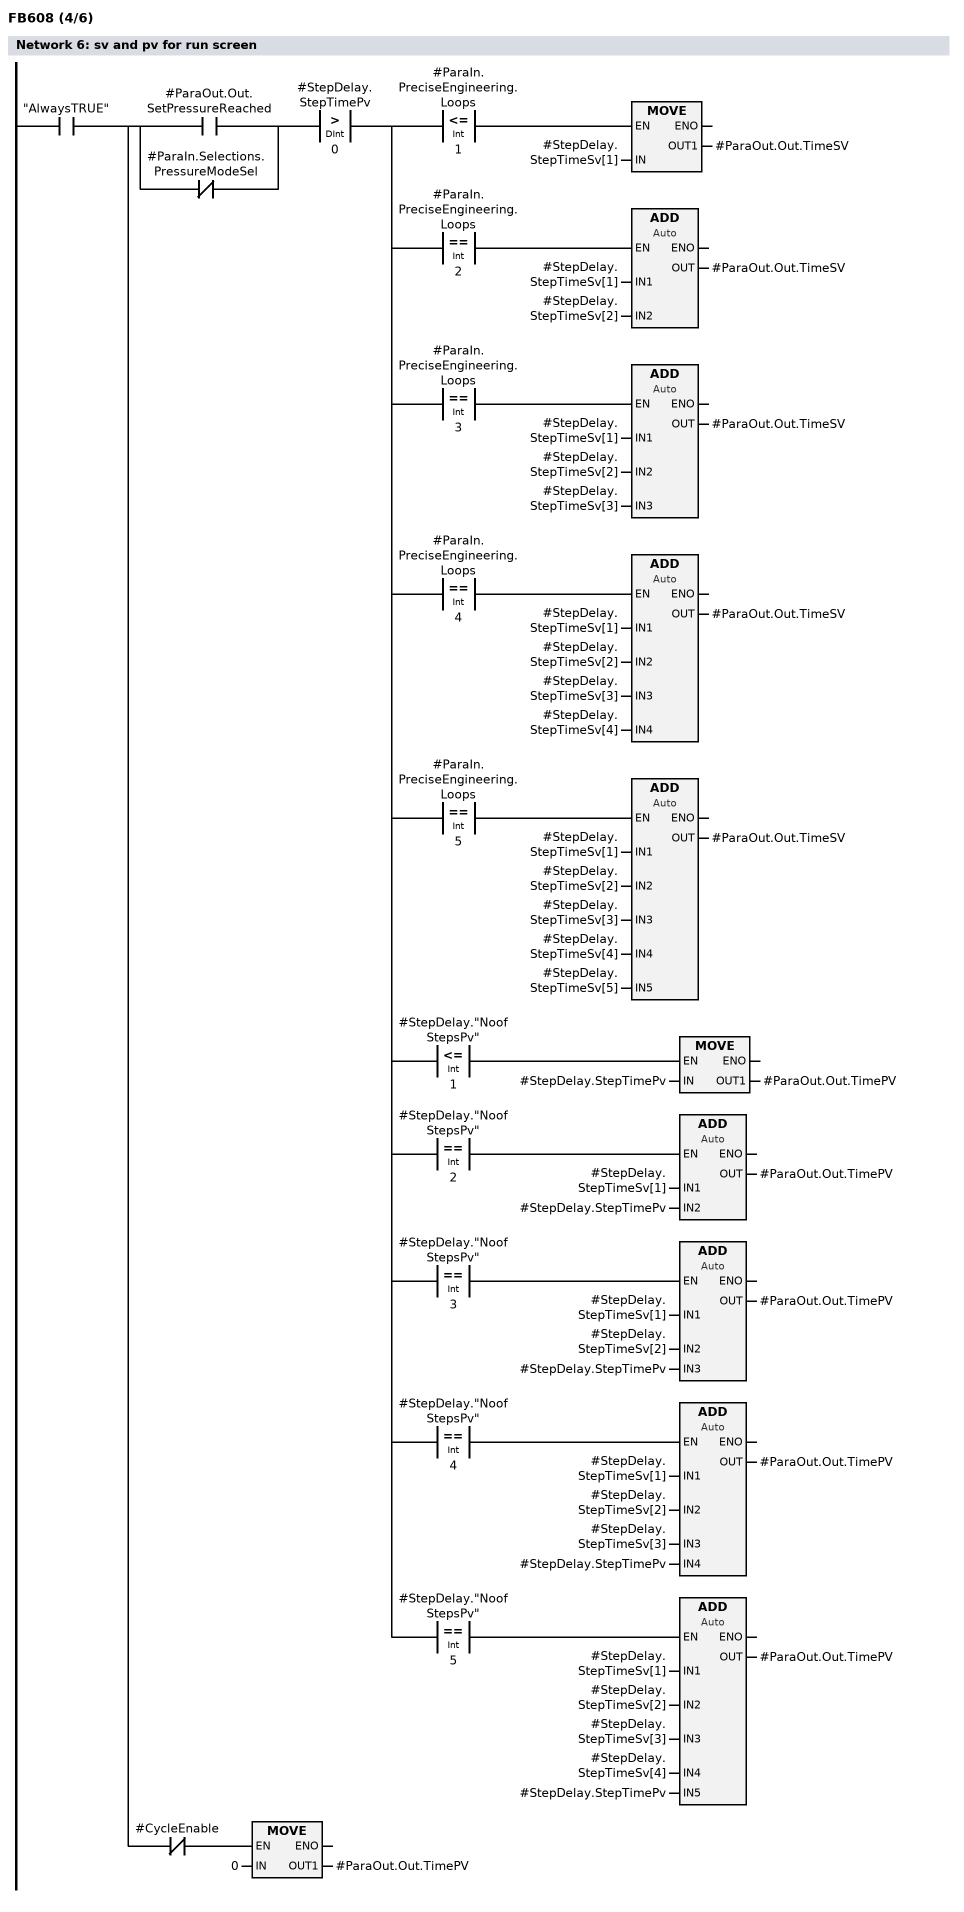
   RUNG wire#powerrail
      Contact( "AlwaysTRUE" )
      wire#w1
      Contact( #ParaOut.Out.SetPressureReached )
      wire#w2
      { S7_Templates := "SrcType := DInt" } GT_Contact(in1 := #StepDelay.StepTimePv, in2 := 0)
      wire#w3
      { S7_Templates := "SrcType := Int" } LE_Contact(in1 := #ParaIn.PreciseEngineering.Loops, in2 := 1)
      Move(in := #StepDelay.StepTimeSv[1], out1 => #ParaOut.Out.TimeSV)
   END_RUNG
   RUNG wire#w1
      I_Contact( #ParaIn.Selections.PressureModeSel )
   END_RUNG wire#w2
   RUNG wire#w3
      { S7_Templates := "SrcType := Int" } EQ_Contact(in1 := #ParaIn.PreciseEngineering.Loops, in2 := 2)
      Add(in1 := #StepDelay.StepTimeSv[1], in2 := #StepDelay.StepTimeSv[2], out => #ParaOut.Out.TimeSV)
   END_RUNG
   RUNG wire#w3
      { S7_Templates := "SrcType := Int" } EQ_Contact(in1 := #ParaIn.PreciseEngineering.Loops, in2 := 3)
      Add(in1 := #StepDelay.StepTimeSv[1], in2 := #StepDelay.StepTimeSv[2], in3 := #StepDelay.StepTimeSv[3], out => #ParaOut.Out.TimeSV)
   END_RUNG
   RUNG wire#w3
      { S7_Templates := "SrcType := Int" } EQ_Contact(in1 := #ParaIn.PreciseEngineering.Loops, in2 := 4)
      Add(in1 := #StepDelay.StepTimeSv[1], in2 := #StepDelay.StepTimeSv[2], in3 := #StepDelay.StepTimeSv[3], in4 := #StepDelay.StepTimeSv[4], out => #ParaOut.Out.TimeSV)
   END_RUNG
   RUNG wire#w3
      { S7_Templates := "SrcType := Int" } EQ_Contact(in1 := #ParaIn.PreciseEngineering.Loops, in2 := 5)
      Add(in1 := #StepDelay.StepTimeSv[1], in2 := #StepDelay.StepTimeSv[2], in3 := #StepDelay.StepTimeSv[3], in4 := #StepDelay.StepTimeSv[4], in5 := #StepDelay.StepTimeSv[5], out => #ParaOut.Out.TimeSV)
   END_RUNG
   RUNG wire#w3
      { S7_Templates := "SrcType := Int" } LE_Contact(in1 := #StepDelay."Noof StepsPv", in2 := 1)
      Move(in := #StepDelay.StepTimePv, out1 => #ParaOut.Out.TimePV)
   END_RUNG
   RUNG wire#w3
      { S7_Templates := "SrcType := Int" } EQ_Contact(in1 := #StepDelay."Noof StepsPv", in2 := 2)
      Add(in1 := #StepDelay.StepTimeSv[1], in2 := #StepDelay.StepTimePv, out => #ParaOut.Out.TimePV)
   END_RUNG
   RUNG wire#w3
      { S7_Templates := "SrcType := Int" } EQ_Contact(in1 := #StepDelay."Noof StepsPv", in2 := 3)
      Add(in1 := #StepDelay.StepTimeSv[1], in2 := #StepDelay.StepTimeSv[2], in3 := #StepDelay.StepTimePv, out => #ParaOut.Out.TimePV)
   END_RUNG
   RUNG wire#w3
      { S7_Templates := "SrcType := Int" } EQ_Contact(in1 := #StepDelay."Noof StepsPv", in2 := 4)
      Add(in1 := #StepDelay.StepTimeSv[1], in2 := #StepDelay.StepTimeSv[2], in3 := #StepDelay.StepTimeSv[3], in4 := #StepDelay.StepTimePv, out => #ParaOut.Out.TimePV)
   END_RUNG
   RUNG wire#w3
      { S7_Templates := "SrcType := Int" } EQ_Contact(in1 := #StepDelay."Noof StepsPv", in2 := 5)
      Add(in1 := #StepDelay.StepTimeSv[1], in2 := #StepDelay.StepTimeSv[2], in3 := #StepDelay.StepTimeSv[3], in4 := #StepDelay.StepTimeSv[4], in5 := #StepDelay.StepTimePv, out => #ParaOut.Out.TimePV)
   END_RUNG
   RUNG wire#w1
      I_Contact( #CycleEnable )
      Move(in := 0, out1 => #ParaOut.Out.TimePV)
   END_RUNG
   // the same network as SCL:
   #_w1 := "AlwaysTRUE" AND (#ParaOut.Out.SetPressureReached OR NOT #ParaIn.Selections.PressureModeSel) AND (#StepDelay.StepTimePv > 0);
   IF #_w1 AND (#ParaIn.PreciseEngineering.Loops <= 1) THEN
       #ParaOut.Out.TimeSV := #StepDelay.StepTimeSv[1];
   END_IF;
   IF #_w1 AND (#ParaIn.PreciseEngineering.Loops = 2) THEN
       #ParaOut.Out.TimeSV := #StepDelay.StepTimeSv[1] + #StepDelay.StepTimeSv[2];
   END_IF;
   IF #_w1 AND (#ParaIn.PreciseEngineering.Loops = 3) THEN
       #ParaOut.Out.TimeSV := #StepDelay.StepTimeSv[1] + #StepDelay.StepTimeSv[2] + #StepDelay.StepTimeSv[3];
   END_IF;
   IF #_w1 AND (#ParaIn.PreciseEngineering.Loops = 4) THEN
       #ParaOut.Out.TimeSV := #StepDelay.StepTimeSv[1] + #StepDelay.StepTimeSv[2] + #StepDelay.StepTimeSv[3] + #StepDelay.StepTimeSv[4];
   END_IF;
   IF #_w1 AND (#ParaIn.PreciseEngineering.Loops = 5) THEN
       #ParaOut.Out.TimeSV := #StepDelay.StepTimeSv[1] + #StepDelay.StepTimeSv[2] + #StepDelay.StepTimeSv[3] + #StepDelay.StepTimeSv[4] + #StepDelay.StepTimeSv[5];
   END_IF;
   IF #_w1 AND (#StepDelay."Noof StepsPv" <= 1) THEN #ParaOut.Out.TimePV := #StepDelay.StepTimePv; END_IF;
   IF #_w1 AND (#StepDelay."Noof StepsPv" = 2) THEN
       #ParaOut.Out.TimePV := #StepDelay.StepTimeSv[1] + #StepDelay.StepTimePv;
   END_IF;
   IF #_w1 AND (#StepDelay."Noof StepsPv" = 3) THEN
       #ParaOut.Out.TimePV := #StepDelay.StepTimeSv[1] + #StepDelay.StepTimeSv[2] + #StepDelay.StepTimePv;
   END_IF;
   IF #_w1 AND (#StepDelay."Noof StepsPv" = 4) THEN
       #ParaOut.Out.TimePV := #StepDelay.StepTimeSv[1] + #StepDelay.StepTimeSv[2] + #StepDelay.StepTimeSv[3] + #StepDelay.StepTimePv;
   END_IF;
   IF #_w1 AND (#StepDelay."Noof StepsPv" = 5) THEN
       #ParaOut.Out.TimePV := #StepDelay.StepTimeSv[1] + #StepDelay.StepTimeSv[2] + #StepDelay.StepTimeSv[3] + #StepDelay.StepTimeSv[4] + #StepDelay.StepTimePv;
   END_IF;
   IF "AlwaysTRUE" AND NOT #CycleEnable THEN #ParaOut.Out.TimePV := 0; END_IF;
END_REGION

REGION Network 7: #StepDelay
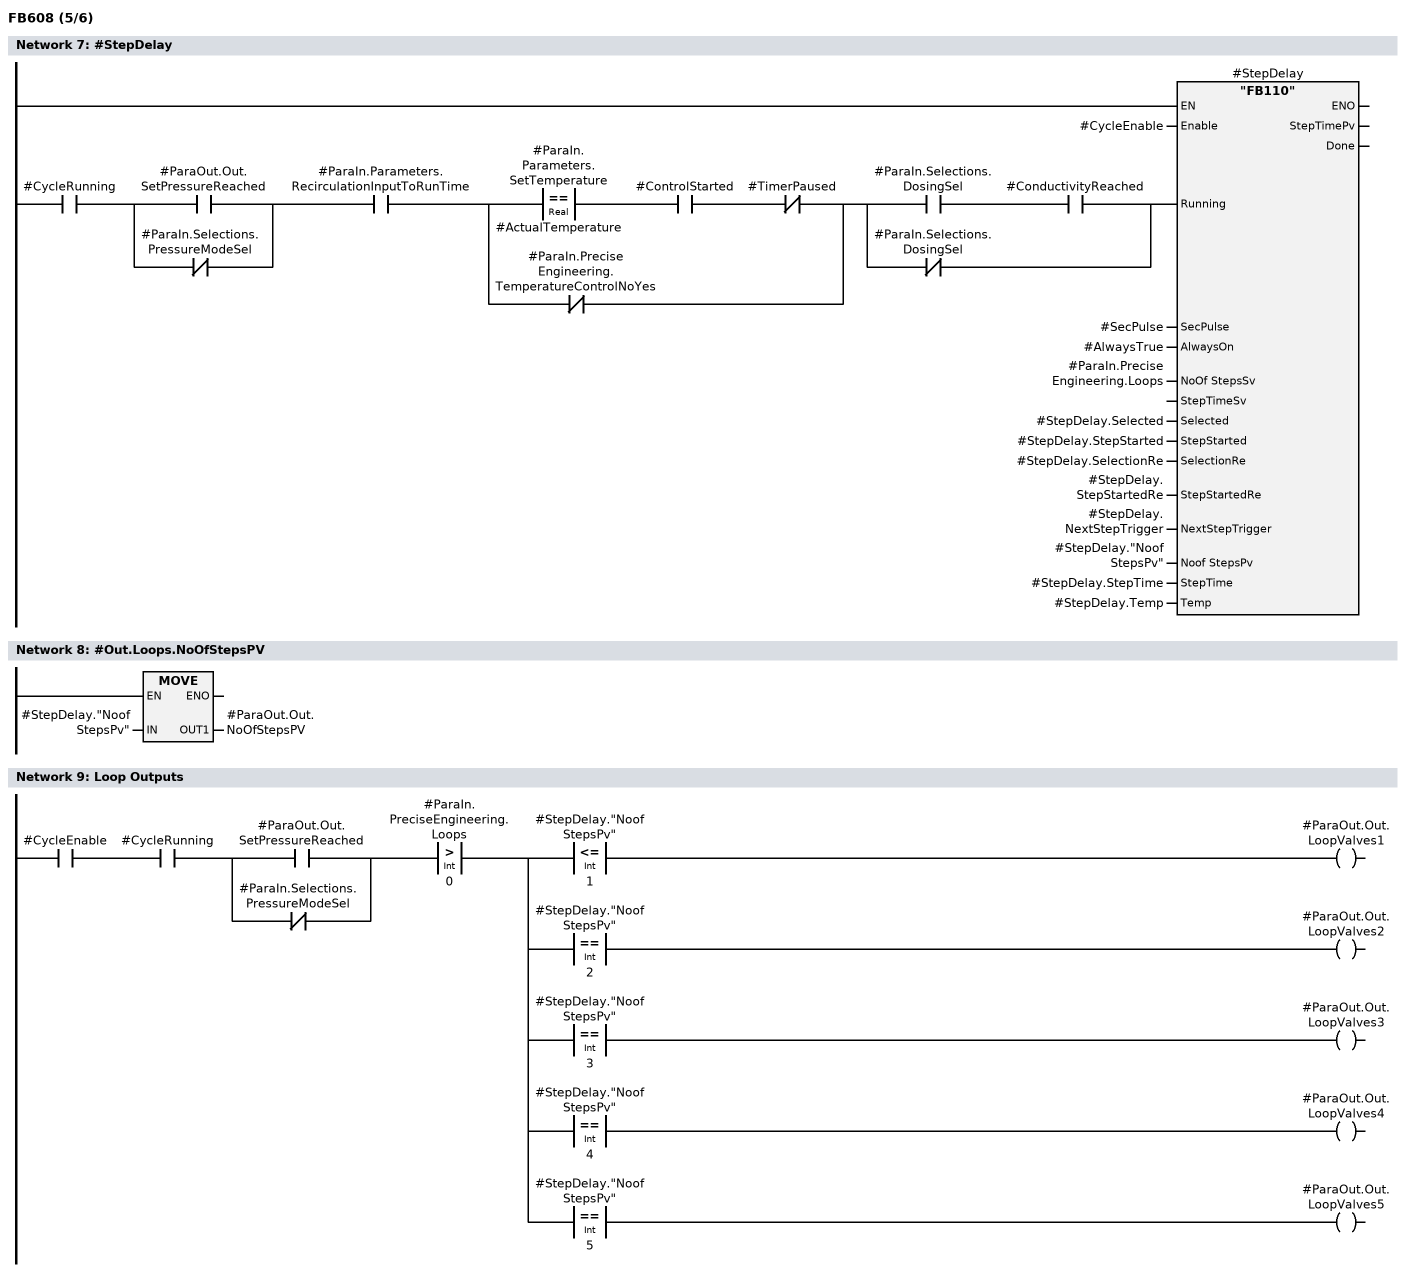
   RUNG wire#powerrail
      #StepDelay(Running := wire#w5, Enable := #CycleEnable, SecPulse := #SecPulse, AlwaysOn := #AlwaysTrue, "NoOf StepsSv" := #ParaIn.PreciseEngineering.Loops, StepTimeSv :=, Selected := #StepDelay.Selected, StepStarted := #StepDelay.StepStarted, SelectionRe := #StepDelay.SelectionRe, StepStartedRe := #StepDelay.StepStartedRe, NextStepTrigger := #StepDelay.NextStepTrigger, "Noof StepsPv" := #StepDelay."Noof StepsPv", StepTime := #StepDelay.StepTime, Temp := #StepDelay.Temp, StepTimePv =>, Done =>)
   END_RUNG
   RUNG wire#powerrail
      Contact( #CycleRunning )
      wire#w1
      Contact( #ParaOut.Out.SetPressureReached )
      wire#w2
      Contact( #ParaIn.Parameters.RecirculationInputToRunTime )
      wire#w3
      { S7_Templates := "SrcType := Real" } EQ_Contact(in1 := #ParaIn.Parameters.SetTemperature, in2 := #ActualTemperature)
      Contact( #ControlStarted )
      I_Contact( #TimerPaused )
      wire#w4
      Contact( #ParaIn.Selections.DosingSel )
      Contact( #ConductivityReached )
   END_RUNG wire#w5
   RUNG wire#w1
      I_Contact( #ParaIn.Selections.PressureModeSel )
   END_RUNG wire#w2
   RUNG wire#w3
      I_Contact( #ParaIn.PreciseEngineering.TemperatureControlNoYes )
   END_RUNG wire#w4
   RUNG wire#w4
      I_Contact( #ParaIn.Selections.DosingSel )
   END_RUNG wire#w5
   // the same network as SCL:
   #StepDelay(Enable := #CycleEnable,   // "FB110"
              Running := #CycleRunning AND (#ParaOut.Out.SetPressureReached OR NOT #ParaIn.Selections.PressureModeSel) AND #ParaIn.Parameters.RecirculationInputToRunTime AND (((#ParaIn.Parameters.SetTemperature = #ActualTemperature) AND #ControlStarted AND NOT #TimerPaused) OR NOT #ParaIn.PreciseEngineering.TemperatureControlNoYes) AND ((#ParaIn.Selections.DosingSel AND #ConductivityReached) OR NOT #ParaIn.Selections.DosingSel),
              SecPulse := #SecPulse,
              AlwaysOn := #AlwaysTrue,
              "NoOf StepsSv" := #ParaIn.PreciseEngineering.Loops,
              Selected := #StepDelay.Selected,
              StepStarted := #StepDelay.StepStarted,
              SelectionRe := #StepDelay.SelectionRe,
              StepStartedRe := #StepDelay.StepStartedRe,
              NextStepTrigger := #StepDelay.NextStepTrigger,
              "Noof StepsPv" := #StepDelay."Noof StepsPv",
              StepTime := #StepDelay.StepTime,
              Temp := #StepDelay.Temp);
END_REGION

REGION Network 8: #Out.Loops.NoOfStepsPV
   RUNG wire#powerrail
      Move(in := #StepDelay."Noof StepsPv", out1 => #ParaOut.Out.NoOfStepsPV)
   END_RUNG
   // the same network as SCL:
   #ParaOut.Out.NoOfStepsPV := #StepDelay."Noof StepsPv";
END_REGION

REGION Network 9: Loop Outputs
   RUNG wire#powerrail
      Contact( #CycleEnable )
      Contact( #CycleRunning )
      wire#w1
      Contact( #ParaOut.Out.SetPressureReached )
      wire#w2
      { S7_Templates := "SrcType := Int" } GT_Contact(in1 := #ParaIn.PreciseEngineering.Loops, in2 := 0)
      wire#w3
      { S7_Templates := "SrcType := Int" } LE_Contact(in1 := #StepDelay."Noof StepsPv", in2 := 1)
      Coil( #ParaOut.Out.LoopValves1 )
   END_RUNG
   RUNG wire#w1
      I_Contact( #ParaIn.Selections.PressureModeSel )
   END_RUNG wire#w2
   RUNG wire#w3
      { S7_Templates := "SrcType := Int" } EQ_Contact(in1 := #StepDelay."Noof StepsPv", in2 := 2)
      Coil( #ParaOut.Out.LoopValves2 )
   END_RUNG
   RUNG wire#w3
      { S7_Templates := "SrcType := Int" } EQ_Contact(in1 := #StepDelay."Noof StepsPv", in2 := 3)
      Coil( #ParaOut.Out.LoopValves3 )
   END_RUNG
   RUNG wire#w3
      { S7_Templates := "SrcType := Int" } EQ_Contact(in1 := #StepDelay."Noof StepsPv", in2 := 4)
      Coil( #ParaOut.Out.LoopValves4 )
   END_RUNG
   RUNG wire#w3
      { S7_Templates := "SrcType := Int" } EQ_Contact(in1 := #StepDelay."Noof StepsPv", in2 := 5)
      Coil( #ParaOut.Out.LoopValves5 )
   END_RUNG
   // the same network as SCL:
   #_w1 := #CycleEnable AND #CycleRunning AND (#ParaOut.Out.SetPressureReached OR NOT #ParaIn.Selections.PressureModeSel) AND (#ParaIn.PreciseEngineering.Loops > 0);
   #ParaOut.Out.LoopValves1 := #_w1 AND (#StepDelay."Noof StepsPv" <= 1);
   #ParaOut.Out.LoopValves2 := #_w1 AND (#StepDelay."Noof StepsPv" = 2);
   #ParaOut.Out.LoopValves3 := #_w1 AND (#StepDelay."Noof StepsPv" = 3);
   #ParaOut.Out.LoopValves4 := #_w1 AND (#StepDelay."Noof StepsPv" = 4);
   #ParaOut.Out.LoopValves5 := #_w1 AND (#StepDelay."Noof StepsPv" = 5);
END_REGION

REGION Network 10: Reset
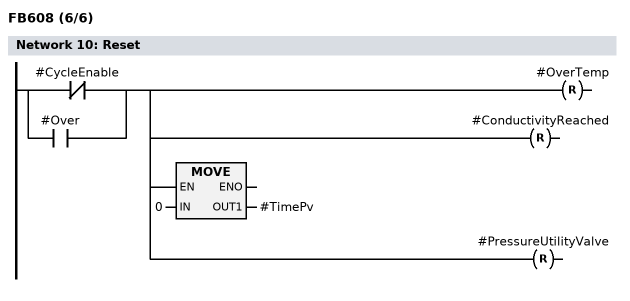
   RUNG wire#powerrail
      I_Contact( #CycleEnable )
      wire#w1
      R_Coil( #OverTemp )
   END_RUNG
   RUNG wire#powerrail
      Contact( #Over )
   END_RUNG wire#w1
   RUNG wire#w1
      R_Coil( #ConductivityReached )
   END_RUNG
   RUNG wire#w1
      { S7_GenerateENO := "TRUE" } Move(in := 0, out1 => #TimePv)
   END_RUNG
   RUNG wire#w1
      R_Coil( #PressureUtilityValve )
   END_RUNG
   // the same network as SCL:
   IF NOT #CycleEnable OR #Over THEN
       #OverTemp := FALSE;
       #ConductivityReached := FALSE;
       #TimePv := 0;
       #PressureUtilityValve := FALSE;
   END_IF;
END_REGION
END_FUNCTION_BLOCK

FUNCTION_BLOCK "FB609"   // FB609, LAD
TITLE = FB609
{ S7_Optimized_Access := 'FALSE' }
AUTHOR : PRECISE
FAMILY : PRECISE
// CIP DRAIN
// stored: AutoNumber false, SetENOAutomatically false
   VAR_INPUT
      CipSelected : Bool;
      CycleEnable : Bool;
      CycleRunning : Bool;
      SecPulse : Bool;
      AlwaysTrue : Bool;
      ParaIn : "DrainInputs";
      ActualWeight : Real;
      ActualPressure : Real;
      ActualConductivityVessel : Real;
      ActualRepetition : Int;
      ActualSkidWeight : Real;
   END_VAR
   VAR_OUTPUT
      Started : Bool;
      PressureUtilityValve : Bool;   // Air Utility
      "Line Valves" : Bool;
      ParaOut : "DrainOutputs";
      StepStatus : String[60];
      Print : "DrainPrint";
      PrintConductivityNotSampled : "ConductivityNotSampled";
   END_VAR
   VAR_IN_OUT
      Over : Bool;
      OverTemp : Bool;
      PressurePostiveTol : Real;
      PressureNegativeTol : Real;
      Temp1 : Int;
      Temp2 : Int;
      SampledConductivityVessel : Real;
      ConductivitySuccess : Bool;
      ConductivityNotSampled : Bool;
      RE1 : Bool;
      RE2 : Bool;
      RE3 : Bool;
      RE4 : Bool;
      RE5 : Bool;
      ControlStarted : Bool;
      SetPressureReached : Bool;
      DrainOverValve : Bool;
      ConductivityCheckBit : Bool;
      ActualConductivityPTL : Real;
      SampledConductivityPTL : Real;
      ConductivitySuccessVessel : Bool;
      ConductivitySuccessPtl : Bool;
      Temp3 : Int;
      Temp4 : Int;
      Temp5 : Int;
      Temp6 : Int;
      Temp7 : Int;
      Temp8 : Int;
      EndConfirmationPopupSel : Bool;
      EndConfirmationPopup : Bool;
      EndConfirmationPopupAck : Bool;
      RE_1 : Bool;
      TempBit : Bool;
      RE6 : Bool;
   END_VAR
   VAR
      ValveOnDelayPV : Int;
      ValveOffDelayPV : Int;
      StepDelay { S7_SetPoint := 'True'} : "FB110";
      ResetPrintValues { S7_SetPoint := 'True'} : TON_TIME;
   END_VAR
   // ParaIn.PreciseEngineering.Loops := 1;
   VAR_TEMP   // added for the SCL form of the ladder/FBD networks
      _w1 : Bool;
      _w2 : Bool;
      _w3 : Bool;
      _w4 : Bool;
      _w5 : Bool;
      _w6 : Bool;
      _w7 : Bool;
      _w8 : Bool;
      _w9 : Bool;
   END_VAR
BEGIN

REGION Network 1: Reset Print Status on Start
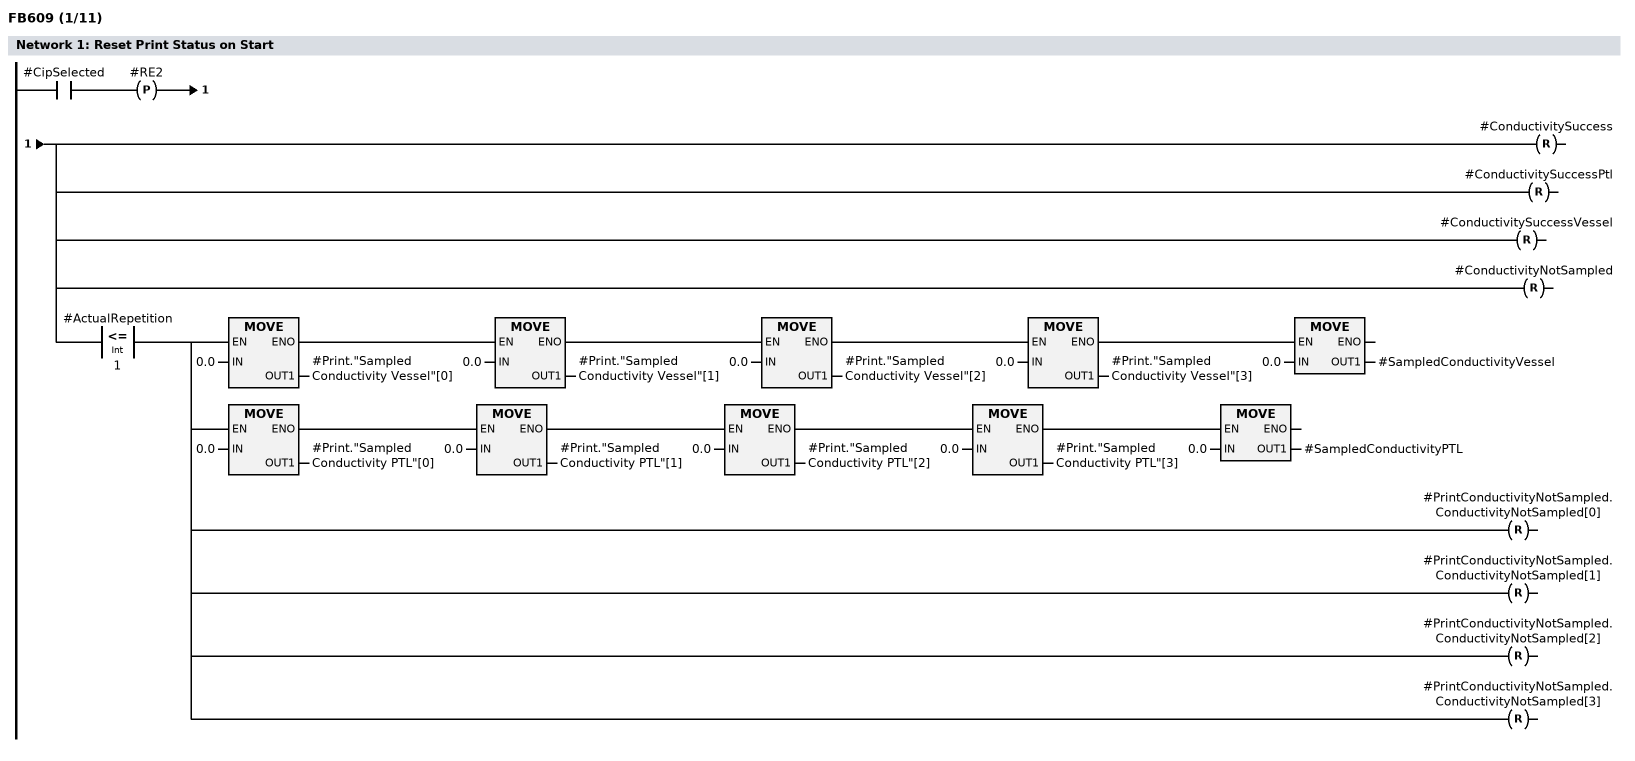
   RUNG wire#powerrail
      Contact( #CipSelected )
      P_Trig( #RE2 )
      wire#w1
      R_Coil( #ConductivitySuccess )
   END_RUNG
   RUNG wire#w1
      R_Coil( #ConductivitySuccessPtl )
   END_RUNG
   RUNG wire#w1
      R_Coil( #ConductivitySuccessVessel )
   END_RUNG
   RUNG wire#w1
      R_Coil( #ConductivityNotSampled )
   END_RUNG
   RUNG wire#w1
      { S7_Templates := "SrcType := Int" } LE_Contact(in1 := #ActualRepetition, in2 := 1)
      wire#w2
      Move(in := 0.0, out1 => #Print."SampledConductivity Vessel"[0])
      Move(in := 0.0, out1 => #Print."SampledConductivity Vessel"[1])
      Move(in := 0.0, out1 => #Print."SampledConductivity Vessel"[2])
      Move(in := 0.0, out1 => #Print."SampledConductivity Vessel"[3])
      Move(in := 0.0, out1 => #SampledConductivityVessel)
   END_RUNG
   RUNG wire#w2
      Move(in := 0.0, out1 => #Print."SampledConductivity PTL"[0])
      Move(in := 0.0, out1 => #Print."SampledConductivity PTL"[1])
      Move(in := 0.0, out1 => #Print."SampledConductivity PTL"[2])
      Move(in := 0.0, out1 => #Print."SampledConductivity PTL"[3])
      Move(in := 0.0, out1 => #SampledConductivityPTL)
   END_RUNG
   RUNG wire#w2
      R_Coil( #PrintConductivityNotSampled.ConductivityNotSampled[0] )
   END_RUNG
   RUNG wire#w2
      R_Coil( #PrintConductivityNotSampled.ConductivityNotSampled[1] )
   END_RUNG
   RUNG wire#w2
      R_Coil( #PrintConductivityNotSampled.ConductivityNotSampled[2] )
   END_RUNG
   RUNG wire#w2
      R_Coil( #PrintConductivityNotSampled.ConductivityNotSampled[3] )
   END_RUNG
   // the same network as SCL:
   #_w1 := #CipSelected AND NOT #RE2;   // rising edge
   #RE2 := #CipSelected;
   IF #_w1 THEN
       #ConductivitySuccess := FALSE;
       #ConductivitySuccessPtl := FALSE;
       #ConductivitySuccessVessel := FALSE;
       #ConductivityNotSampled := FALSE;
   END_IF;
   IF #_w1 AND (#ActualRepetition <= 1) THEN
       #Print."SampledConductivity Vessel"[0] := 0.0;
       #Print."SampledConductivity Vessel"[1] := 0.0;
       #Print."SampledConductivity Vessel"[2] := 0.0;
       #Print."SampledConductivity Vessel"[3] := 0.0;
       #SampledConductivityVessel := 0.0;
       #Print."SampledConductivity PTL"[0] := 0.0;
       #Print."SampledConductivity PTL"[1] := 0.0;
       #Print."SampledConductivity PTL"[2] := 0.0;
       #Print."SampledConductivity PTL"[3] := 0.0;
       #SampledConductivityPTL := 0.0;
       #PrintConductivityNotSampled.ConductivityNotSampled[0] := FALSE;
       #PrintConductivityNotSampled.ConductivityNotSampled[1] := FALSE;
       #PrintConductivityNotSampled.ConductivityNotSampled[2] := FALSE;
       #PrintConductivityNotSampled.ConductivityNotSampled[3] := FALSE;
   END_IF;
END_REGION

REGION Network 2: Drain Started
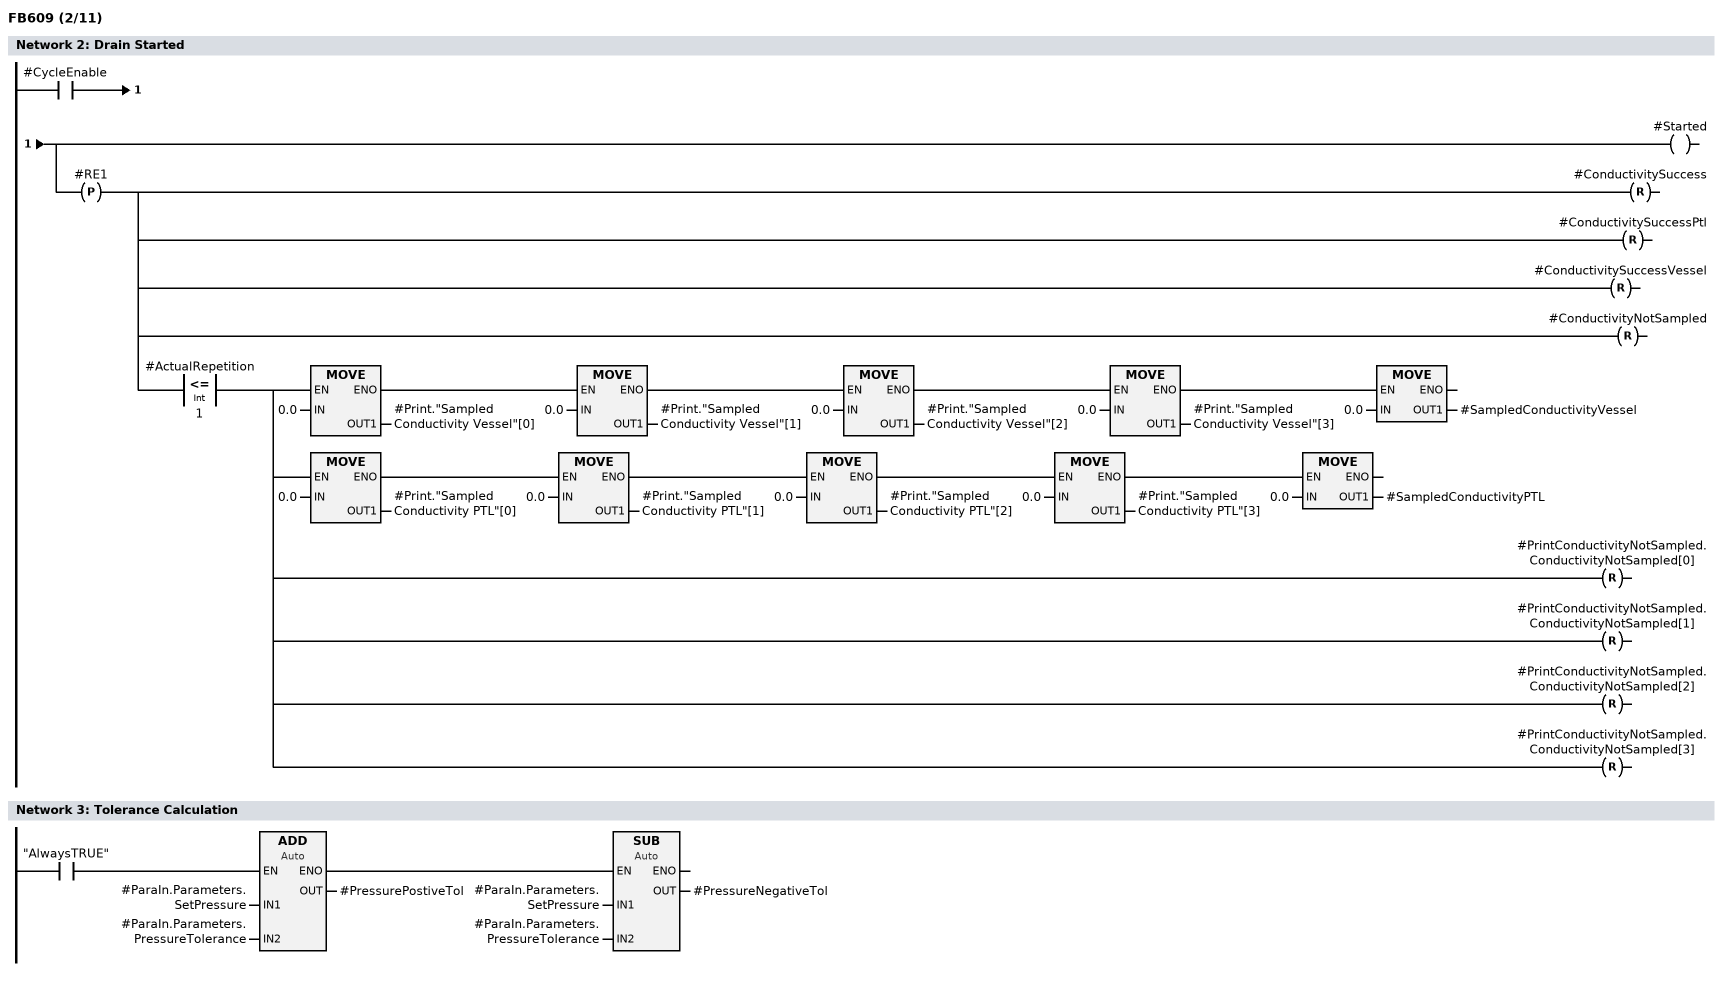
   RUNG wire#powerrail
      Contact( #CycleEnable )
      wire#w1
      Coil( #Started )
   END_RUNG
   RUNG wire#w1
      P_Trig( #RE1 )
      wire#w2
      R_Coil( #ConductivitySuccess )
   END_RUNG
   RUNG wire#w2
      R_Coil( #ConductivitySuccessPtl )
   END_RUNG
   RUNG wire#w2
      R_Coil( #ConductivitySuccessVessel )
   END_RUNG
   RUNG wire#w2
      R_Coil( #ConductivityNotSampled )
   END_RUNG
   RUNG wire#w2
      { S7_Templates := "SrcType := Int" } LE_Contact(in1 := #ActualRepetition, in2 := 1)
      wire#w3
      Move(in := 0.0, out1 => #Print."SampledConductivity Vessel"[0])
      Move(in := 0.0, out1 => #Print."SampledConductivity Vessel"[1])
      Move(in := 0.0, out1 => #Print."SampledConductivity Vessel"[2])
      Move(in := 0.0, out1 => #Print."SampledConductivity Vessel"[3])
      Move(in := 0.0, out1 => #SampledConductivityVessel)
   END_RUNG
   RUNG wire#w3
      Move(in := 0.0, out1 => #Print."SampledConductivity PTL"[0])
      Move(in := 0.0, out1 => #Print."SampledConductivity PTL"[1])
      Move(in := 0.0, out1 => #Print."SampledConductivity PTL"[2])
      Move(in := 0.0, out1 => #Print."SampledConductivity PTL"[3])
      Move(in := 0.0, out1 => #SampledConductivityPTL)
   END_RUNG
   RUNG wire#w3
      R_Coil( #PrintConductivityNotSampled.ConductivityNotSampled[0] )
   END_RUNG
   RUNG wire#w3
      R_Coil( #PrintConductivityNotSampled.ConductivityNotSampled[1] )
   END_RUNG
   RUNG wire#w3
      R_Coil( #PrintConductivityNotSampled.ConductivityNotSampled[2] )
   END_RUNG
   RUNG wire#w3
      R_Coil( #PrintConductivityNotSampled.ConductivityNotSampled[3] )
   END_RUNG
   // the same network as SCL:
   #Started := #CycleEnable;
   #_w1 := #CycleEnable AND NOT #RE1;   // rising edge
   #RE1 := #CycleEnable;
   IF #_w1 THEN
       #ConductivitySuccess := FALSE;
       #ConductivitySuccessPtl := FALSE;
       #ConductivitySuccessVessel := FALSE;
       #ConductivityNotSampled := FALSE;
   END_IF;
   IF #_w1 AND (#ActualRepetition <= 1) THEN
       #Print."SampledConductivity Vessel"[0] := 0.0;
       #Print."SampledConductivity Vessel"[1] := 0.0;
       #Print."SampledConductivity Vessel"[2] := 0.0;
       #Print."SampledConductivity Vessel"[3] := 0.0;
       #SampledConductivityVessel := 0.0;
       #Print."SampledConductivity PTL"[0] := 0.0;
       #Print."SampledConductivity PTL"[1] := 0.0;
       #Print."SampledConductivity PTL"[2] := 0.0;
       #Print."SampledConductivity PTL"[3] := 0.0;
       #SampledConductivityPTL := 0.0;
       #PrintConductivityNotSampled.ConductivityNotSampled[0] := FALSE;
       #PrintConductivityNotSampled.ConductivityNotSampled[1] := FALSE;
       #PrintConductivityNotSampled.ConductivityNotSampled[2] := FALSE;
       #PrintConductivityNotSampled.ConductivityNotSampled[3] := FALSE;
   END_IF;
END_REGION

REGION Network 3: Tolerance Calculation
   RUNG wire#powerrail
      Contact( "AlwaysTRUE" )
      Add(in1 := #ParaIn.Parameters.SetPressure, in2 := #ParaIn.Parameters.PressureTolerance, out => #PressurePostiveTol)
      Sub(in1 := #ParaIn.Parameters.SetPressure, in2 := #ParaIn.Parameters.PressureTolerance, out => #PressureNegativeTol)
   END_RUNG
   // the same network as SCL:
   IF "AlwaysTRUE" THEN
       #PressurePostiveTol := #ParaIn.Parameters.SetPressure + #ParaIn.Parameters.PressureTolerance;
       #PressureNegativeTol := #ParaIn.Parameters.SetPressure - #ParaIn.Parameters.PressureTolerance;
   END_IF;
END_REGION

REGION Network 4: Logic for Output
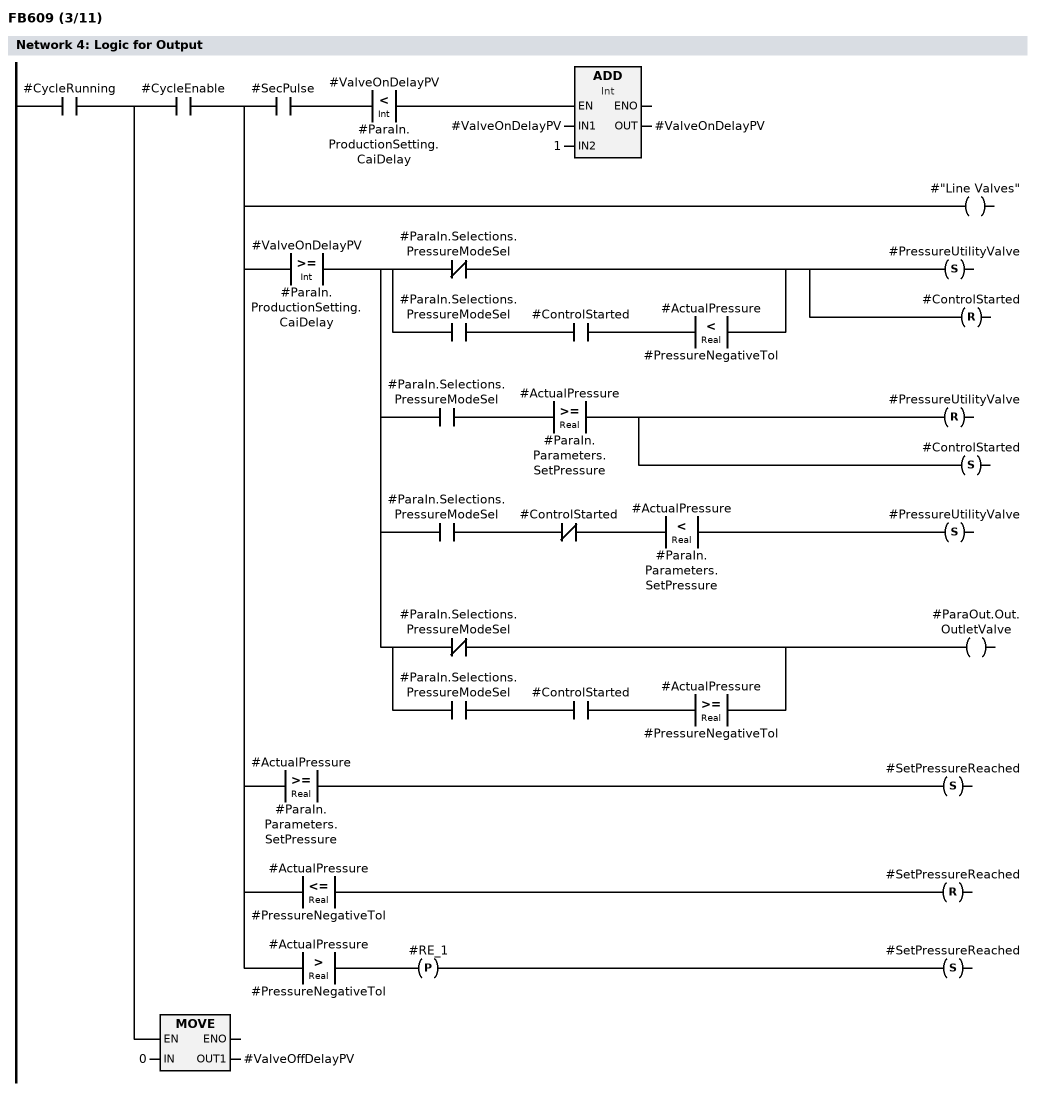
   RUNG wire#powerrail
      Contact( #CycleRunning )
      wire#w1
      Contact( #CycleEnable )
      wire#w2
      Contact( #SecPulse )
      { S7_Templates := "SrcType := Int" } LT_Contact(in1 := #ValveOnDelayPV, in2 := #ParaIn.ProductionSetting.CaiDelay)
      { S7_Templates := "SrcType := Int"; S7_GenerateENO := "TRUE" } Add(in1 := #ValveOnDelayPV, in2 := 1, out => #ValveOnDelayPV)
   END_RUNG
   RUNG wire#w2
      Coil( #"Line Valves" )
   END_RUNG
   RUNG wire#w2
      { S7_Templates := "SrcType := Int" } GE_Contact(in1 := #ValveOnDelayPV, in2 := #ParaIn.ProductionSetting.CaiDelay)
      wire#w3
      I_Contact( #ParaIn.Selections.PressureModeSel )
      wire#w4
      S_Coil( #PressureUtilityValve )
   END_RUNG
   RUNG wire#w3
      Contact( #ParaIn.Selections.PressureModeSel )
      Contact( #ControlStarted )
      { S7_Templates := "SrcType := Real" } LT_Contact(in1 := #ActualPressure, in2 := #PressureNegativeTol)
   END_RUNG wire#w4
   RUNG wire#w4
      R_Coil( #ControlStarted )
   END_RUNG
   RUNG wire#w3
      Contact( #ParaIn.Selections.PressureModeSel )
      { S7_Templates := "SrcType := Real" } GE_Contact(in1 := #ActualPressure, in2 := #ParaIn.Parameters.SetPressure)
      wire#w5
      R_Coil( #PressureUtilityValve )
   END_RUNG
   RUNG wire#w5
      S_Coil( #ControlStarted )
   END_RUNG
   RUNG wire#w3
      Contact( #ParaIn.Selections.PressureModeSel )
      I_Contact( #ControlStarted )
      { S7_Templates := "SrcType := Real" } LT_Contact(in1 := #ActualPressure, in2 := #ParaIn.Parameters.SetPressure)
      S_Coil( #PressureUtilityValve )
   END_RUNG
   RUNG wire#w3
      I_Contact( #ParaIn.Selections.PressureModeSel )
      wire#w6
      Coil( #ParaOut.Out.OutletValve )
   END_RUNG
   RUNG wire#w3
      Contact( #ParaIn.Selections.PressureModeSel )
      Contact( #ControlStarted )
      { S7_Templates := "SrcType := Real" } GE_Contact(in1 := #ActualPressure, in2 := #PressureNegativeTol)
   END_RUNG wire#w6
   RUNG wire#w2
      { S7_Templates := "SrcType := Real" } GE_Contact(in1 := #ActualPressure, in2 := #ParaIn.Parameters.SetPressure)
      S_Coil( #SetPressureReached )
   END_RUNG
   RUNG wire#w2
      { S7_Templates := "SrcType := Real" } LE_Contact(in1 := #ActualPressure, in2 := #PressureNegativeTol)
      R_Coil( #SetPressureReached )
   END_RUNG
   RUNG wire#w2
      { S7_Templates := "SrcType := Real" } GT_Contact(in1 := #ActualPressure, in2 := #PressureNegativeTol)
      P_Trig( #RE_1 )
      S_Coil( #SetPressureReached )
   END_RUNG
   RUNG wire#w1
      { S7_GenerateENO := "TRUE" } Move(in := 0, out1 => #ValveOffDelayPV)
   END_RUNG
   // the same network as SCL:
   #_w1 := #CycleRunning AND #CycleEnable;
   IF #_w1 AND #SecPulse AND (#ValveOnDelayPV < #ParaIn.ProductionSetting.CaiDelay) THEN
       #ValveOnDelayPV := #ValveOnDelayPV + 1;
   END_IF;
   #"Line Valves" := #_w1;
   #_w2 := #_w1 AND (#ValveOnDelayPV >= #ParaIn.ProductionSetting.CaiDelay);
   IF #_w2 AND (NOT #ParaIn.Selections.PressureModeSel OR (#ParaIn.Selections.PressureModeSel AND #ControlStarted AND (#ActualPressure < #PressureNegativeTol))) THEN
       #PressureUtilityValve := TRUE;
       #ControlStarted := FALSE;
   END_IF;
   IF #_w2 AND #ParaIn.Selections.PressureModeSel AND (#ActualPressure >= #ParaIn.Parameters.SetPressure) THEN
       #PressureUtilityValve := FALSE;
       #ControlStarted := TRUE;
   END_IF;
   IF #_w2 AND #ParaIn.Selections.PressureModeSel AND NOT #ControlStarted AND (#ActualPressure < #ParaIn.Parameters.SetPressure) THEN
       #PressureUtilityValve := TRUE;
   END_IF;
   #ParaOut.Out.OutletValve := #_w2 AND (NOT #ParaIn.Selections.PressureModeSel OR (#ParaIn.Selections.PressureModeSel AND #ControlStarted AND (#ActualPressure >= #PressureNegativeTol)));
   IF #_w1 AND (#ActualPressure >= #ParaIn.Parameters.SetPressure) THEN #SetPressureReached := TRUE; END_IF;
   IF #_w1 AND (#ActualPressure <= #PressureNegativeTol) THEN #SetPressureReached := FALSE; END_IF;
   #_w3 := #_w1 AND (#ActualPressure > #PressureNegativeTol);
   #_w4 := #_w3 AND NOT #RE_1;   // rising edge
   #RE_1 := #_w3;
   IF #_w4 THEN #SetPressureReached := TRUE; END_IF;
   IF #CycleRunning THEN #ValveOffDelayPV := 0; END_IF;
END_REGION

REGION Network 5: Drain Over Condition
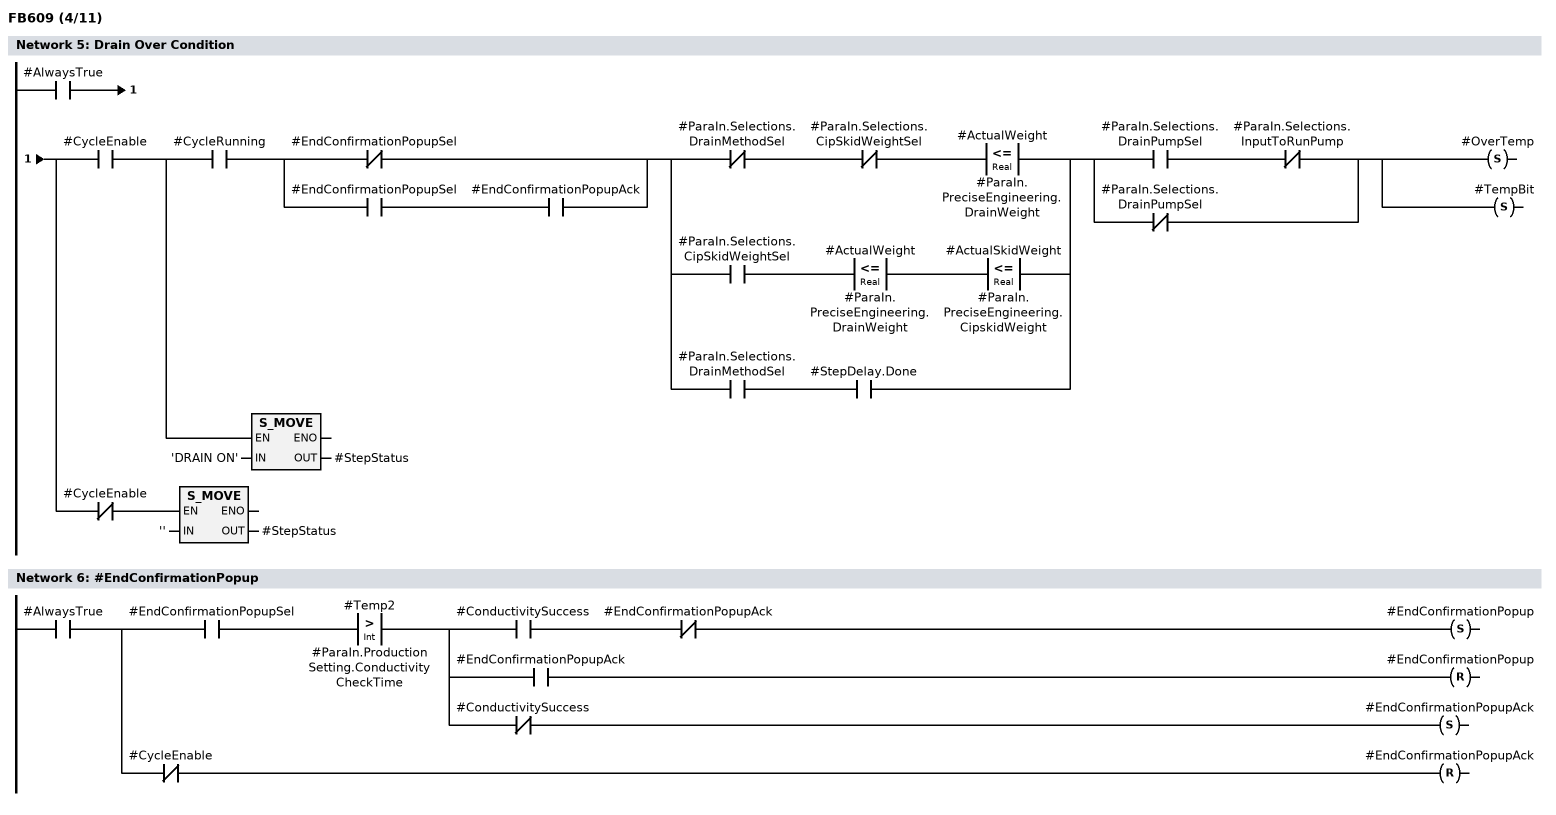
   RUNG wire#powerrail
      Contact( #AlwaysTrue )
      wire#w1
      Contact( #CycleEnable )
      wire#w2
      Contact( #CycleRunning )
      wire#w3
      I_Contact( #EndConfirmationPopupSel )
      wire#w4
      I_Contact( #ParaIn.Selections.DrainMethodSel )
      I_Contact( #ParaIn.Selections.CipSkidWeightSel )
      { S7_Templates := "SrcType := Real" } LE_Contact(in1 := #ActualWeight, in2 := #ParaIn.PreciseEngineering.DrainWeight)
      wire#w5
      Contact( #ParaIn.Selections.DrainPumpSel )
      I_Contact( #ParaIn.Selections.InputToRunPump )
      wire#w6
      S_Coil( #OverTemp )
   END_RUNG
   RUNG wire#w3
      Contact( #EndConfirmationPopupSel )
      Contact( #EndConfirmationPopupAck )
   END_RUNG wire#w4
   RUNG wire#w4
      Contact( #ParaIn.Selections.CipSkidWeightSel )
      { S7_Templates := "SrcType := Real" } LE_Contact(in1 := #ActualWeight, in2 := #ParaIn.PreciseEngineering.DrainWeight)
      { S7_Templates := "SrcType := Real" } LE_Contact(in1 := #ActualSkidWeight, in2 := #ParaIn.PreciseEngineering.CipskidWeight)
   END_RUNG wire#w5
   RUNG wire#w4
      Contact( #ParaIn.Selections.DrainMethodSel )
      Contact( #StepDelay.Done )
   END_RUNG wire#w5
   RUNG wire#w5
      I_Contact( #ParaIn.Selections.DrainPumpSel )
   END_RUNG wire#w6
   RUNG wire#w6
      S_Coil( #TempBit )
   END_RUNG
   RUNG wire#w2
      S_Move(in := 'DRAIN ON', out => #StepStatus)
   END_RUNG
   RUNG wire#w1
      I_Contact( #CycleEnable )
      S_Move(in := '', out => #StepStatus)
   END_RUNG
   // the same network as SCL:
   #_w1 := #AlwaysTrue AND #CycleEnable;
   IF #_w1 AND #CycleRunning AND (NOT #EndConfirmationPopupSel OR (#EndConfirmationPopupSel AND #EndConfirmationPopupAck)) AND ((NOT #ParaIn.Selections.DrainMethodSel AND NOT #ParaIn.Selections.CipSkidWeightSel AND (#ActualWeight <= #ParaIn.PreciseEngineering.DrainWeight)) OR (#ParaIn.Selections.CipSkidWeightSel AND (#ActualWeight <= #ParaIn.PreciseEngineering.DrainWeight) AND (#ActualSkidWeight <= #ParaIn.PreciseEngineering.CipskidWeight)) OR (#ParaIn.Selections.DrainMethodSel AND #StepDelay.Done)) AND ((#ParaIn.Selections.DrainPumpSel AND NOT #ParaIn.Selections.InputToRunPump) OR NOT #ParaIn.Selections.DrainPumpSel) THEN
       #OverTemp := TRUE;
       #TempBit := TRUE;
   END_IF;
   IF #_w1 THEN #StepStatus := 'DRAIN ON'; END_IF;
   IF #AlwaysTrue AND NOT #CycleEnable THEN #StepStatus := ''; END_IF;
END_REGION

REGION Network 6: #EndConfirmationPopup
   RUNG wire#powerrail
      Contact( #AlwaysTrue )
      wire#w1
      Contact( #EndConfirmationPopupSel )
      { S7_Templates := "SrcType := Int" } GT_Contact(in1 := #Temp2, in2 := #ParaIn.ProductionSetting.ConductivityCheckTime)
      wire#w2
      Contact( #ConductivitySuccess )
      I_Contact( #EndConfirmationPopupAck )
      S_Coil( #EndConfirmationPopup )
   END_RUNG
   RUNG wire#w2
      Contact( #EndConfirmationPopupAck )
      R_Coil( #EndConfirmationPopup )
   END_RUNG
   RUNG wire#w2
      I_Contact( #ConductivitySuccess )
      S_Coil( #EndConfirmationPopupAck )
   END_RUNG
   RUNG wire#w1
      I_Contact( #CycleEnable )
      R_Coil( #EndConfirmationPopupAck )
   END_RUNG
   // the same network as SCL:
   #_w1 := #AlwaysTrue AND #EndConfirmationPopupSel AND (#Temp2 > #ParaIn.ProductionSetting.ConductivityCheckTime);
   IF #_w1 AND #ConductivitySuccess AND NOT #EndConfirmationPopupAck THEN
       #EndConfirmationPopup := TRUE;
   END_IF;
   IF #_w1 AND #EndConfirmationPopupAck THEN #EndConfirmationPopup := FALSE; END_IF;
   IF #_w1 AND NOT #ConductivitySuccess THEN #EndConfirmationPopupAck := TRUE; END_IF;
   IF #AlwaysTrue AND NOT #CycleEnable THEN #EndConfirmationPopupAck := FALSE; END_IF;
END_REGION

REGION Network 7: Air Purge Over
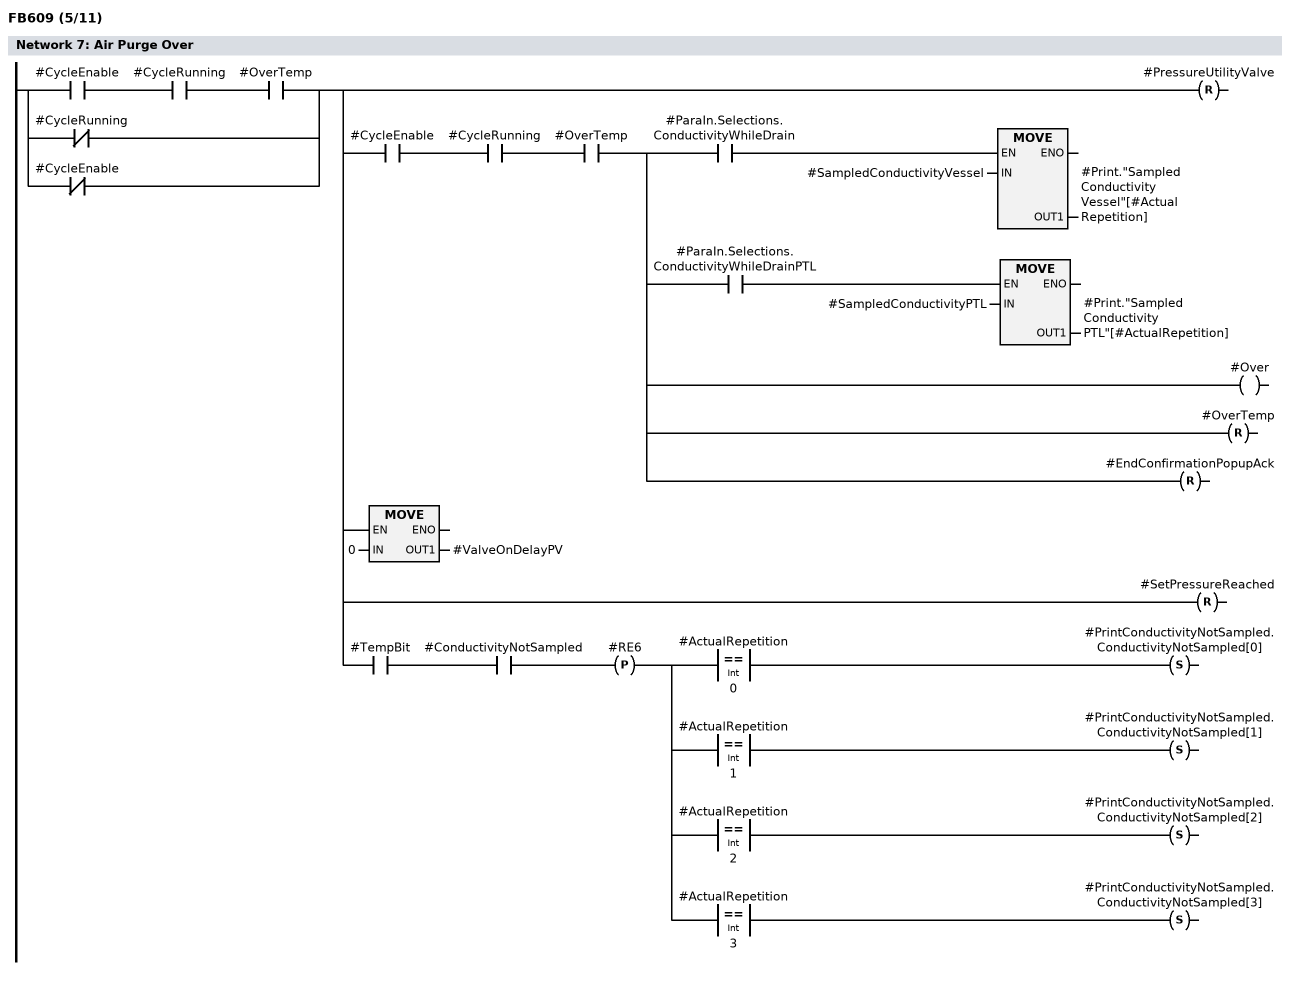
   RUNG wire#powerrail
      Contact( #CycleEnable )
      Contact( #CycleRunning )
      Contact( #OverTemp )
      wire#w1
      R_Coil( #PressureUtilityValve )
   END_RUNG
   RUNG wire#powerrail
      I_Contact( #CycleRunning )
   END_RUNG wire#w1
   RUNG wire#powerrail
      I_Contact( #CycleEnable )
   END_RUNG wire#w1
   RUNG wire#w1
      Contact( #CycleEnable )
      Contact( #CycleRunning )
      Contact( #OverTemp )
      wire#w2
      Contact( #ParaIn.Selections.ConductivityWhileDrain )
      Move(in := #SampledConductivityVessel, out1 => #Print."SampledConductivity Vessel"[#ActualRepetition])
   END_RUNG
   RUNG wire#w2
      Contact( #ParaIn.Selections.ConductivityWhileDrainPTL )
      Move(in := #SampledConductivityPTL, out1 => #Print."SampledConductivity PTL"[#ActualRepetition])
   END_RUNG
   RUNG wire#w2
      Coil( #Over )
   END_RUNG
   RUNG wire#w2
      R_Coil( #OverTemp )
   END_RUNG
   RUNG wire#w2
      R_Coil( #EndConfirmationPopupAck )
   END_RUNG
   RUNG wire#w1
      Move(in := 0, out1 => #ValveOnDelayPV)
   END_RUNG
   RUNG wire#w1
      R_Coil( #SetPressureReached )
   END_RUNG
   RUNG wire#w1
      Contact( #TempBit )
      Contact( #ConductivityNotSampled )
      P_Trig( #RE6 )
      wire#w3
      { S7_Templates := "SrcType := Int" } EQ_Contact(in1 := #ActualRepetition, in2 := 0)
      S_Coil( #PrintConductivityNotSampled.ConductivityNotSampled[0] )
   END_RUNG
   RUNG wire#w3
      { S7_Templates := "SrcType := Int" } EQ_Contact(in1 := #ActualRepetition, in2 := 1)
      S_Coil( #PrintConductivityNotSampled.ConductivityNotSampled[1] )
   END_RUNG
   RUNG wire#w3
      { S7_Templates := "SrcType := Int" } EQ_Contact(in1 := #ActualRepetition, in2 := 2)
      S_Coil( #PrintConductivityNotSampled.ConductivityNotSampled[2] )
   END_RUNG
   RUNG wire#w3
      { S7_Templates := "SrcType := Int" } EQ_Contact(in1 := #ActualRepetition, in2 := 3)
      S_Coil( #PrintConductivityNotSampled.ConductivityNotSampled[3] )
   END_RUNG
   // the same network as SCL:
   #_w1 := (#CycleEnable AND #CycleRunning AND #OverTemp) OR NOT #CycleRunning OR NOT #CycleEnable;
   IF #_w1 THEN #PressureUtilityValve := FALSE; END_IF;
   #_w2 := #_w1 AND #CycleEnable AND #CycleRunning AND #OverTemp;
   IF #_w2 AND #ParaIn.Selections.ConductivityWhileDrain THEN
       #Print."SampledConductivity Vessel"[#ActualRepetition] := #SampledConductivityVessel;
   END_IF;
   IF #_w2 AND #ParaIn.Selections.ConductivityWhileDrainPTL THEN
       #Print."SampledConductivity PTL"[#ActualRepetition] := #SampledConductivityPTL;
   END_IF;
   #Over := #_w2;
   IF #_w2 THEN
       #OverTemp := FALSE;
       #EndConfirmationPopupAck := FALSE;
   END_IF;
   IF #_w1 THEN
       #ValveOnDelayPV := 0;
       #SetPressureReached := FALSE;
   END_IF;
   #_w3 := #_w1 AND #TempBit AND #ConductivityNotSampled;
   #_w4 := #_w3 AND NOT #RE6;   // rising edge
   #RE6 := #_w3;
   IF #_w4 AND (#ActualRepetition = 0) THEN
       #PrintConductivityNotSampled.ConductivityNotSampled[0] := TRUE;
   END_IF;
   IF #_w4 AND (#ActualRepetition = 1) THEN
       #PrintConductivityNotSampled.ConductivityNotSampled[1] := TRUE;
   END_IF;
   IF #_w4 AND (#ActualRepetition = 2) THEN
       #PrintConductivityNotSampled.ConductivityNotSampled[2] := TRUE;
   END_IF;
   IF #_w4 AND (#ActualRepetition = 3) THEN
       #PrintConductivityNotSampled.ConductivityNotSampled[3] := TRUE;
   END_IF;
END_REGION

REGION Network 8: StepDelay.StepTimeSV
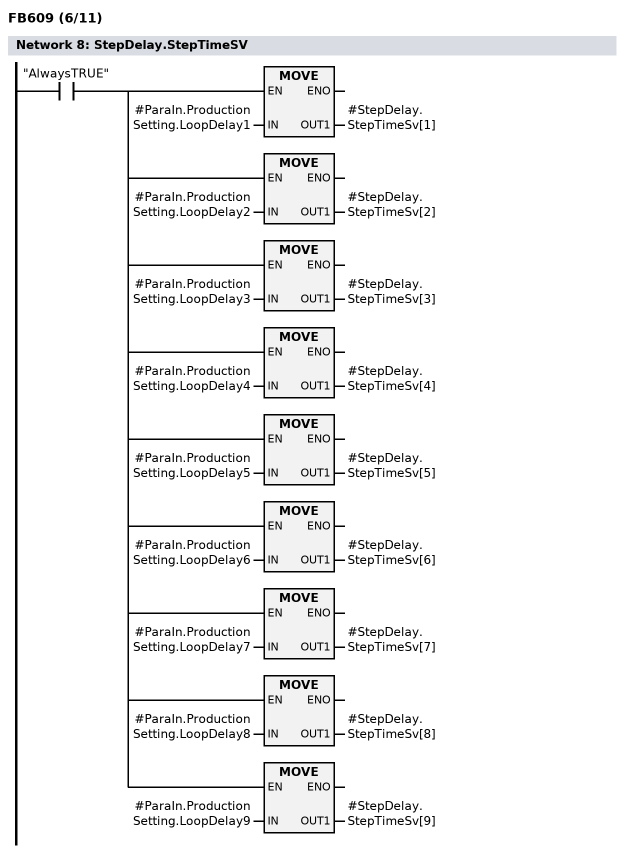
   RUNG wire#powerrail
      Contact( "AlwaysTRUE" )
      wire#w1
      Move(in := #ParaIn.ProductionSetting.LoopDelay1, out1 => #StepDelay.StepTimeSv[1])
   END_RUNG
   RUNG wire#w1
      Move(in := #ParaIn.ProductionSetting.LoopDelay2, out1 => #StepDelay.StepTimeSv[2])
   END_RUNG
   RUNG wire#w1
      Move(in := #ParaIn.ProductionSetting.LoopDelay3, out1 => #StepDelay.StepTimeSv[3])
   END_RUNG
   RUNG wire#w1
      Move(in := #ParaIn.ProductionSetting.LoopDelay4, out1 => #StepDelay.StepTimeSv[4])
   END_RUNG
   RUNG wire#w1
      Move(in := #ParaIn.ProductionSetting.LoopDelay5, out1 => #StepDelay.StepTimeSv[5])
   END_RUNG
   RUNG wire#w1
      Move(in := #ParaIn.ProductionSetting.LoopDelay6, out1 => #StepDelay.StepTimeSv[6])
   END_RUNG
   RUNG wire#w1
      Move(in := #ParaIn.ProductionSetting.LoopDelay7, out1 => #StepDelay.StepTimeSv[7])
   END_RUNG
   RUNG wire#w1
      Move(in := #ParaIn.ProductionSetting.LoopDelay8, out1 => #StepDelay.StepTimeSv[8])
   END_RUNG
   RUNG wire#w1
      Move(in := #ParaIn.ProductionSetting.LoopDelay9, out1 => #StepDelay.StepTimeSv[9])
   END_RUNG
   // the same network as SCL:
   IF "AlwaysTRUE" THEN
       #StepDelay.StepTimeSv[1] := #ParaIn.ProductionSetting.LoopDelay1;
       #StepDelay.StepTimeSv[2] := #ParaIn.ProductionSetting.LoopDelay2;
       #StepDelay.StepTimeSv[3] := #ParaIn.ProductionSetting.LoopDelay3;
       #StepDelay.StepTimeSv[4] := #ParaIn.ProductionSetting.LoopDelay4;
       #StepDelay.StepTimeSv[5] := #ParaIn.ProductionSetting.LoopDelay5;
       #StepDelay.StepTimeSv[6] := #ParaIn.ProductionSetting.LoopDelay6;
       #StepDelay.StepTimeSv[7] := #ParaIn.ProductionSetting.LoopDelay7;
       #StepDelay.StepTimeSv[8] := #ParaIn.ProductionSetting.LoopDelay8;
       #StepDelay.StepTimeSv[9] := #ParaIn.ProductionSetting.LoopDelay9;
   END_IF;
END_REGION

REGION Network 9: #StepDelay
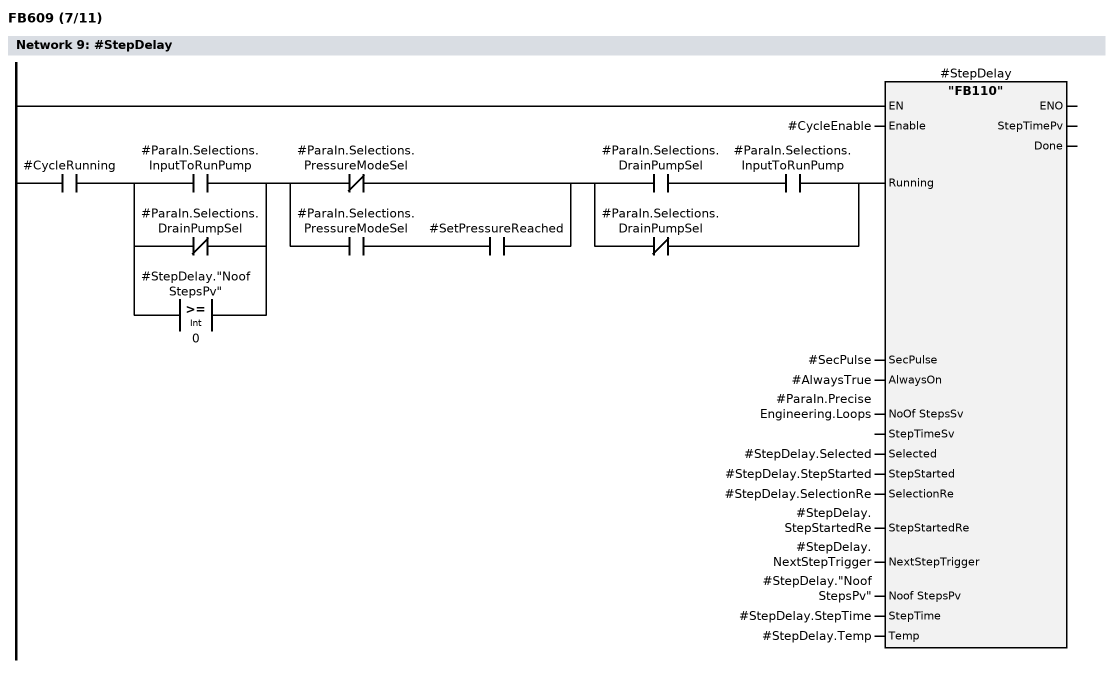
   RUNG wire#powerrail
      #StepDelay(Running := wire#w4, Enable := #CycleEnable, SecPulse := #SecPulse, AlwaysOn := #AlwaysTrue, "NoOf StepsSv" := #ParaIn.PreciseEngineering.Loops, StepTimeSv :=, Selected := #StepDelay.Selected, StepStarted := #StepDelay.StepStarted, SelectionRe := #StepDelay.SelectionRe, StepStartedRe := #StepDelay.StepStartedRe, NextStepTrigger := #StepDelay.NextStepTrigger, "Noof StepsPv" := #StepDelay."Noof StepsPv", StepTime := #StepDelay.StepTime, Temp := #StepDelay.Temp, StepTimePv =>, Done =>)
   END_RUNG
   RUNG wire#powerrail
      Contact( #CycleRunning )
      wire#w1
      Contact( #ParaIn.Selections.InputToRunPump )
      wire#w2
      I_Contact( #ParaIn.Selections.PressureModeSel )
      wire#w3
      Contact( #ParaIn.Selections.DrainPumpSel )
      Contact( #ParaIn.Selections.InputToRunPump )
   END_RUNG wire#w4
   RUNG wire#w1
      I_Contact( #ParaIn.Selections.DrainPumpSel )
   END_RUNG wire#w2
   RUNG wire#w1
      { S7_Templates := "SrcType := Int" } GE_Contact(in1 := #StepDelay."Noof StepsPv", in2 := 0)
   END_RUNG wire#w2
   RUNG wire#w2
      Contact( #ParaIn.Selections.PressureModeSel )
      Contact( #SetPressureReached )
   END_RUNG wire#w3
   RUNG wire#w3
      I_Contact( #ParaIn.Selections.DrainPumpSel )
   END_RUNG wire#w4
   // the same network as SCL:
   #StepDelay(Enable := #CycleEnable,   // "FB110"
              Running := #CycleRunning AND (#ParaIn.Selections.InputToRunPump OR NOT #ParaIn.Selections.DrainPumpSel OR (#StepDelay."Noof StepsPv" >= 0)) AND (NOT #ParaIn.Selections.PressureModeSel OR (#ParaIn.Selections.PressureModeSel AND #SetPressureReached)) AND ((#ParaIn.Selections.DrainPumpSel AND #ParaIn.Selections.InputToRunPump) OR NOT #ParaIn.Selections.DrainPumpSel),
              SecPulse := #SecPulse,
              AlwaysOn := #AlwaysTrue,
              "NoOf StepsSv" := #ParaIn.PreciseEngineering.Loops,
              Selected := #StepDelay.Selected,
              StepStarted := #StepDelay.StepStarted,
              SelectionRe := #StepDelay.SelectionRe,
              StepStartedRe := #StepDelay.StepStartedRe,
              NextStepTrigger := #StepDelay.NextStepTrigger,
              "Noof StepsPv" := #StepDelay."Noof StepsPv",
              StepTime := #StepDelay.StepTime,
              Temp := #StepDelay.Temp);
END_REGION

REGION Network 10: Loop Outputs
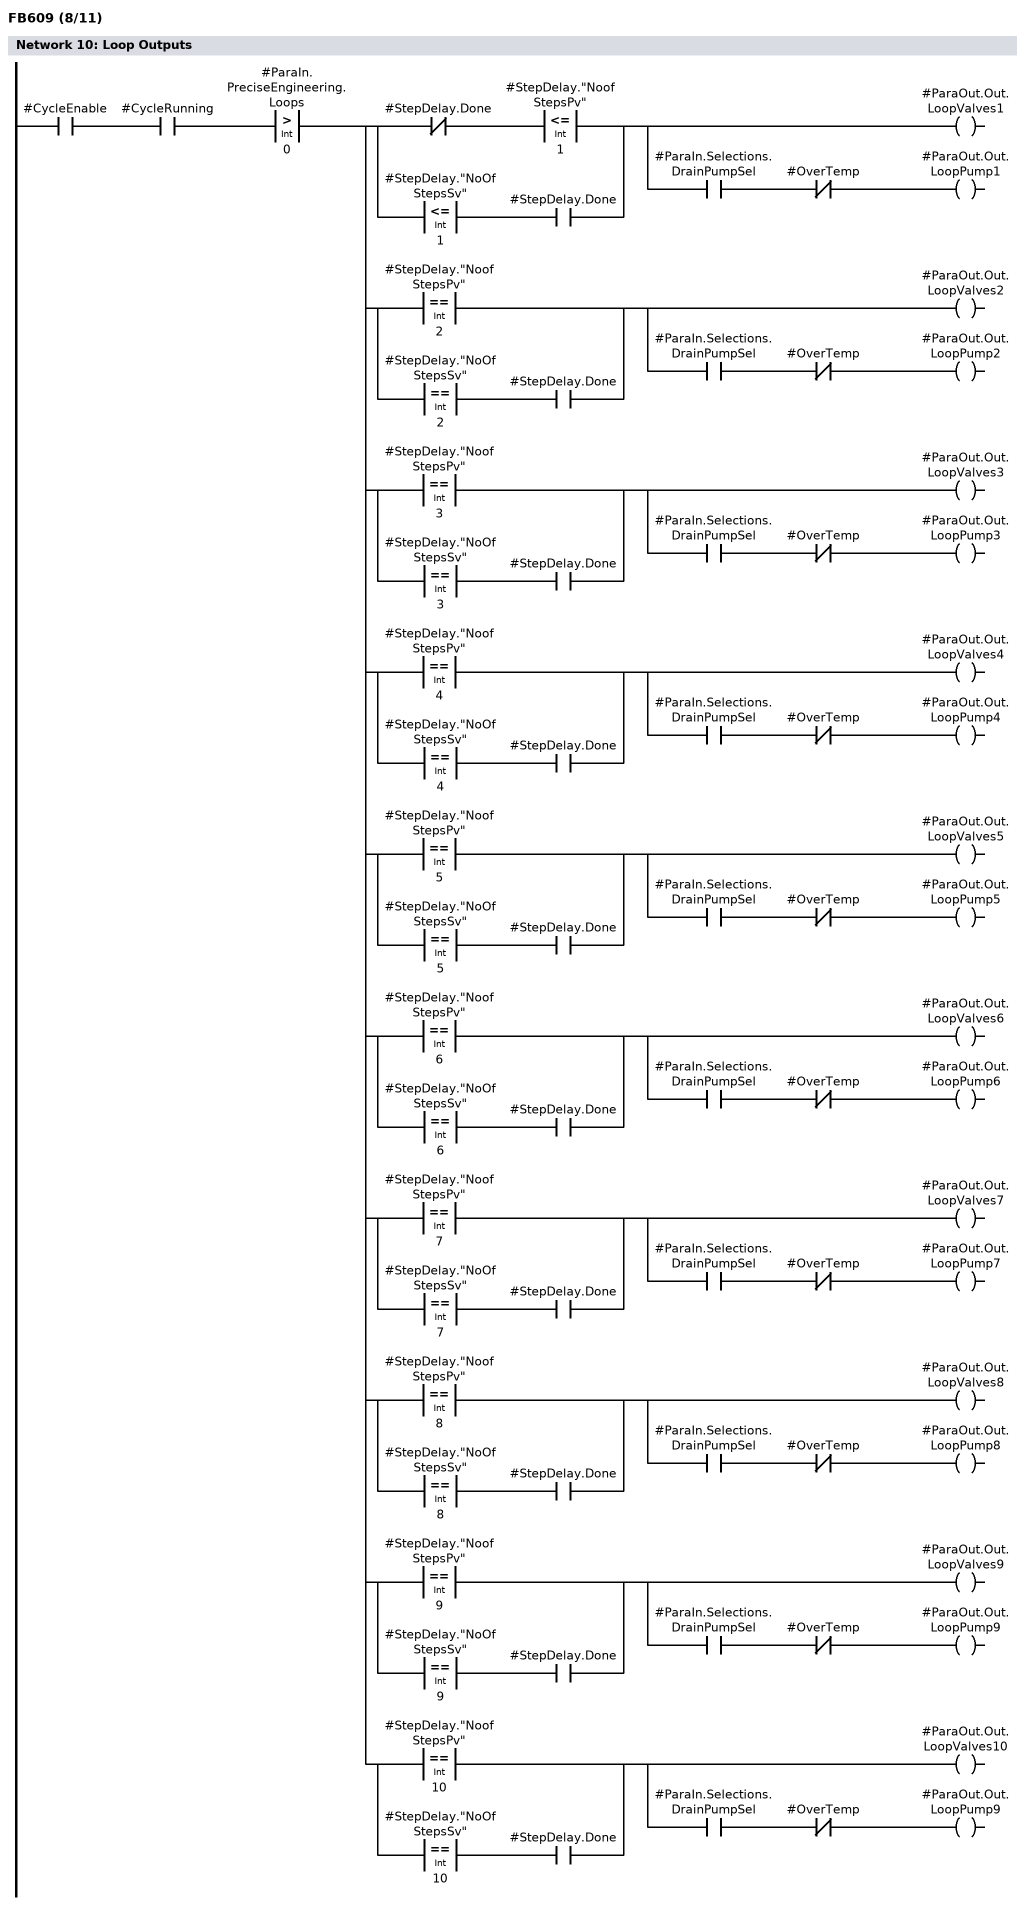
   RUNG wire#powerrail
      Contact( #CycleEnable )
      Contact( #CycleRunning )
      { S7_Templates := "SrcType := Int" } GT_Contact(in1 := #ParaIn.PreciseEngineering.Loops, in2 := 0)
      wire#w1
      I_Contact( #StepDelay.Done )
      { S7_Templates := "SrcType := Int" } LE_Contact(in1 := #StepDelay."Noof StepsPv", in2 := 1)
      wire#w2
      Coil( #ParaOut.Out.LoopValves1 )
   END_RUNG
   RUNG wire#w1
      { S7_Templates := "SrcType := Int" } LE_Contact(in1 := #StepDelay."NoOf StepsSv", in2 := 1)
      Contact( #StepDelay.Done )
   END_RUNG wire#w2
   RUNG wire#w2
      Contact( #ParaIn.Selections.DrainPumpSel )
      I_Contact( #OverTemp )
      Coil( #ParaOut.Out.LoopPump1 )
   END_RUNG
   RUNG wire#w1
      { S7_Templates := "SrcType := Int" } EQ_Contact(in1 := #StepDelay."Noof StepsPv", in2 := 2)
      wire#w3
      Coil( #ParaOut.Out.LoopValves2 )
   END_RUNG
   RUNG wire#w1
      { S7_Templates := "SrcType := Int" } EQ_Contact(in1 := #StepDelay."NoOf StepsSv", in2 := 2)
      Contact( #StepDelay.Done )
   END_RUNG wire#w3
   RUNG wire#w3
      Contact( #ParaIn.Selections.DrainPumpSel )
      I_Contact( #OverTemp )
      Coil( #ParaOut.Out.LoopPump2 )
   END_RUNG
   RUNG wire#w1
      { S7_Templates := "SrcType := Int" } EQ_Contact(in1 := #StepDelay."Noof StepsPv", in2 := 3)
      wire#w4
      Coil( #ParaOut.Out.LoopValves3 )
   END_RUNG
   RUNG wire#w1
      { S7_Templates := "SrcType := Int" } EQ_Contact(in1 := #StepDelay."NoOf StepsSv", in2 := 3)
      Contact( #StepDelay.Done )
   END_RUNG wire#w4
   RUNG wire#w4
      Contact( #ParaIn.Selections.DrainPumpSel )
      I_Contact( #OverTemp )
      Coil( #ParaOut.Out.LoopPump3 )
   END_RUNG
   RUNG wire#w1
      { S7_Templates := "SrcType := Int" } EQ_Contact(in1 := #StepDelay."Noof StepsPv", in2 := 4)
      wire#w5
      Coil( #ParaOut.Out.LoopValves4 )
   END_RUNG
   RUNG wire#w1
      { S7_Templates := "SrcType := Int" } EQ_Contact(in1 := #StepDelay."NoOf StepsSv", in2 := 4)
      Contact( #StepDelay.Done )
   END_RUNG wire#w5
   RUNG wire#w5
      Contact( #ParaIn.Selections.DrainPumpSel )
      I_Contact( #OverTemp )
      Coil( #ParaOut.Out.LoopPump4 )
   END_RUNG
   RUNG wire#w1
      { S7_Templates := "SrcType := Int" } EQ_Contact(in1 := #StepDelay."Noof StepsPv", in2 := 5)
      wire#w6
      Coil( #ParaOut.Out.LoopValves5 )
   END_RUNG
   RUNG wire#w1
      { S7_Templates := "SrcType := Int" } EQ_Contact(in1 := #StepDelay."NoOf StepsSv", in2 := 5)
      Contact( #StepDelay.Done )
   END_RUNG wire#w6
   RUNG wire#w6
      Contact( #ParaIn.Selections.DrainPumpSel )
      I_Contact( #OverTemp )
      Coil( #ParaOut.Out.LoopPump5 )
   END_RUNG
   RUNG wire#w1
      { S7_Templates := "SrcType := Int" } EQ_Contact(in1 := #StepDelay."Noof StepsPv", in2 := 6)
      wire#w7
      Coil( #ParaOut.Out.LoopValves6 )
   END_RUNG
   RUNG wire#w1
      { S7_Templates := "SrcType := Int" } EQ_Contact(in1 := #StepDelay."NoOf StepsSv", in2 := 6)
      Contact( #StepDelay.Done )
   END_RUNG wire#w7
   RUNG wire#w7
      Contact( #ParaIn.Selections.DrainPumpSel )
      I_Contact( #OverTemp )
      Coil( #ParaOut.Out.LoopPump6 )
   END_RUNG
   RUNG wire#w1
      { S7_Templates := "SrcType := Int" } EQ_Contact(in1 := #StepDelay."Noof StepsPv", in2 := 7)
      wire#w8
      Coil( #ParaOut.Out.LoopValves7 )
   END_RUNG
   RUNG wire#w1
      { S7_Templates := "SrcType := Int" } EQ_Contact(in1 := #StepDelay."NoOf StepsSv", in2 := 7)
      Contact( #StepDelay.Done )
   END_RUNG wire#w8
   RUNG wire#w8
      Contact( #ParaIn.Selections.DrainPumpSel )
      I_Contact( #OverTemp )
      Coil( #ParaOut.Out.LoopPump7 )
   END_RUNG
   RUNG wire#w1
      { S7_Templates := "SrcType := Int" } EQ_Contact(in1 := #StepDelay."Noof StepsPv", in2 := 8)
      wire#w9
      Coil( #ParaOut.Out.LoopValves8 )
   END_RUNG
   RUNG wire#w1
      { S7_Templates := "SrcType := Int" } EQ_Contact(in1 := #StepDelay."NoOf StepsSv", in2 := 8)
      Contact( #StepDelay.Done )
   END_RUNG wire#w9
   RUNG wire#w9
      Contact( #ParaIn.Selections.DrainPumpSel )
      I_Contact( #OverTemp )
      Coil( #ParaOut.Out.LoopPump8 )
   END_RUNG
   RUNG wire#w1
      { S7_Templates := "SrcType := Int" } EQ_Contact(in1 := #StepDelay."Noof StepsPv", in2 := 9)
      wire#w10
      Coil( #ParaOut.Out.LoopValves9 )
   END_RUNG
   RUNG wire#w1
      { S7_Templates := "SrcType := Int" } EQ_Contact(in1 := #StepDelay."NoOf StepsSv", in2 := 9)
      Contact( #StepDelay.Done )
   END_RUNG wire#w10
   RUNG wire#w10
      Contact( #ParaIn.Selections.DrainPumpSel )
      I_Contact( #OverTemp )
      Coil( #ParaOut.Out.LoopPump9 )
   END_RUNG
   RUNG wire#w1
      { S7_Templates := "SrcType := Int" } EQ_Contact(in1 := #StepDelay."Noof StepsPv", in2 := 10)
      wire#w11
      Coil( #ParaOut.Out.LoopValves10 )
   END_RUNG
   RUNG wire#w1
      { S7_Templates := "SrcType := Int" } EQ_Contact(in1 := #StepDelay."NoOf StepsSv", in2 := 10)
      Contact( #StepDelay.Done )
   END_RUNG wire#w11
   RUNG wire#w11
      Contact( #ParaIn.Selections.DrainPumpSel )
      I_Contact( #OverTemp )
      Coil( #ParaOut.Out.LoopPump9 )
   END_RUNG
   // the same network as SCL:
   #_w1 := #CycleEnable AND #CycleRunning AND (#ParaIn.PreciseEngineering.Loops > 0);
   #ParaOut.Out.LoopValves1 := #_w1 AND ((NOT #StepDelay.Done AND (#StepDelay."Noof StepsPv" <= 1)) OR ((#StepDelay."NoOf StepsSv" <= 1) AND #StepDelay.Done));
   #ParaOut.Out.LoopPump1 := #ParaOut.Out.LoopValves1 AND #ParaIn.Selections.DrainPumpSel AND NOT #OverTemp;
   #ParaOut.Out.LoopValves2 := #_w1 AND ((#StepDelay."Noof StepsPv" = 2) OR ((#StepDelay."NoOf StepsSv" = 2) AND #StepDelay.Done));
   #ParaOut.Out.LoopPump2 := #ParaOut.Out.LoopValves2 AND #ParaIn.Selections.DrainPumpSel AND NOT #OverTemp;
   #ParaOut.Out.LoopValves3 := #_w1 AND ((#StepDelay."Noof StepsPv" = 3) OR ((#StepDelay."NoOf StepsSv" = 3) AND #StepDelay.Done));
   #ParaOut.Out.LoopPump3 := #ParaOut.Out.LoopValves3 AND #ParaIn.Selections.DrainPumpSel AND NOT #OverTemp;
   #ParaOut.Out.LoopValves4 := #_w1 AND ((#StepDelay."Noof StepsPv" = 4) OR ((#StepDelay."NoOf StepsSv" = 4) AND #StepDelay.Done));
   #ParaOut.Out.LoopPump4 := #ParaOut.Out.LoopValves4 AND #ParaIn.Selections.DrainPumpSel AND NOT #OverTemp;
   #ParaOut.Out.LoopValves5 := #_w1 AND ((#StepDelay."Noof StepsPv" = 5) OR ((#StepDelay."NoOf StepsSv" = 5) AND #StepDelay.Done));
   #ParaOut.Out.LoopPump5 := #ParaOut.Out.LoopValves5 AND #ParaIn.Selections.DrainPumpSel AND NOT #OverTemp;
   #ParaOut.Out.LoopValves6 := #_w1 AND ((#StepDelay."Noof StepsPv" = 6) OR ((#StepDelay."NoOf StepsSv" = 6) AND #StepDelay.Done));
   #ParaOut.Out.LoopPump6 := #ParaOut.Out.LoopValves6 AND #ParaIn.Selections.DrainPumpSel AND NOT #OverTemp;
   #ParaOut.Out.LoopValves7 := #_w1 AND ((#StepDelay."Noof StepsPv" = 7) OR ((#StepDelay."NoOf StepsSv" = 7) AND #StepDelay.Done));
   #ParaOut.Out.LoopPump7 := #ParaOut.Out.LoopValves7 AND #ParaIn.Selections.DrainPumpSel AND NOT #OverTemp;
   #ParaOut.Out.LoopValves8 := #_w1 AND ((#StepDelay."Noof StepsPv" = 8) OR ((#StepDelay."NoOf StepsSv" = 8) AND #StepDelay.Done));
   #ParaOut.Out.LoopPump8 := #ParaOut.Out.LoopValves8 AND #ParaIn.Selections.DrainPumpSel AND NOT #OverTemp;
   #ParaOut.Out.LoopValves9 := #_w1 AND ((#StepDelay."Noof StepsPv" = 9) OR ((#StepDelay."NoOf StepsSv" = 9) AND #StepDelay.Done));
   #ParaOut.Out.LoopPump9 := #ParaOut.Out.LoopValves9 AND #ParaIn.Selections.DrainPumpSel AND NOT #OverTemp;
   #ParaOut.Out.LoopValves10 := #_w1 AND ((#StepDelay."Noof StepsPv" = 10) OR ((#StepDelay."NoOf StepsSv" = 10) AND #StepDelay.Done));
   #ParaOut.Out.LoopPump9 := #ParaOut.Out.LoopValves10 AND #ParaIn.Selections.DrainPumpSel AND NOT #OverTemp;
END_REGION

REGION Network 11: Conductivity- Single Conductivity
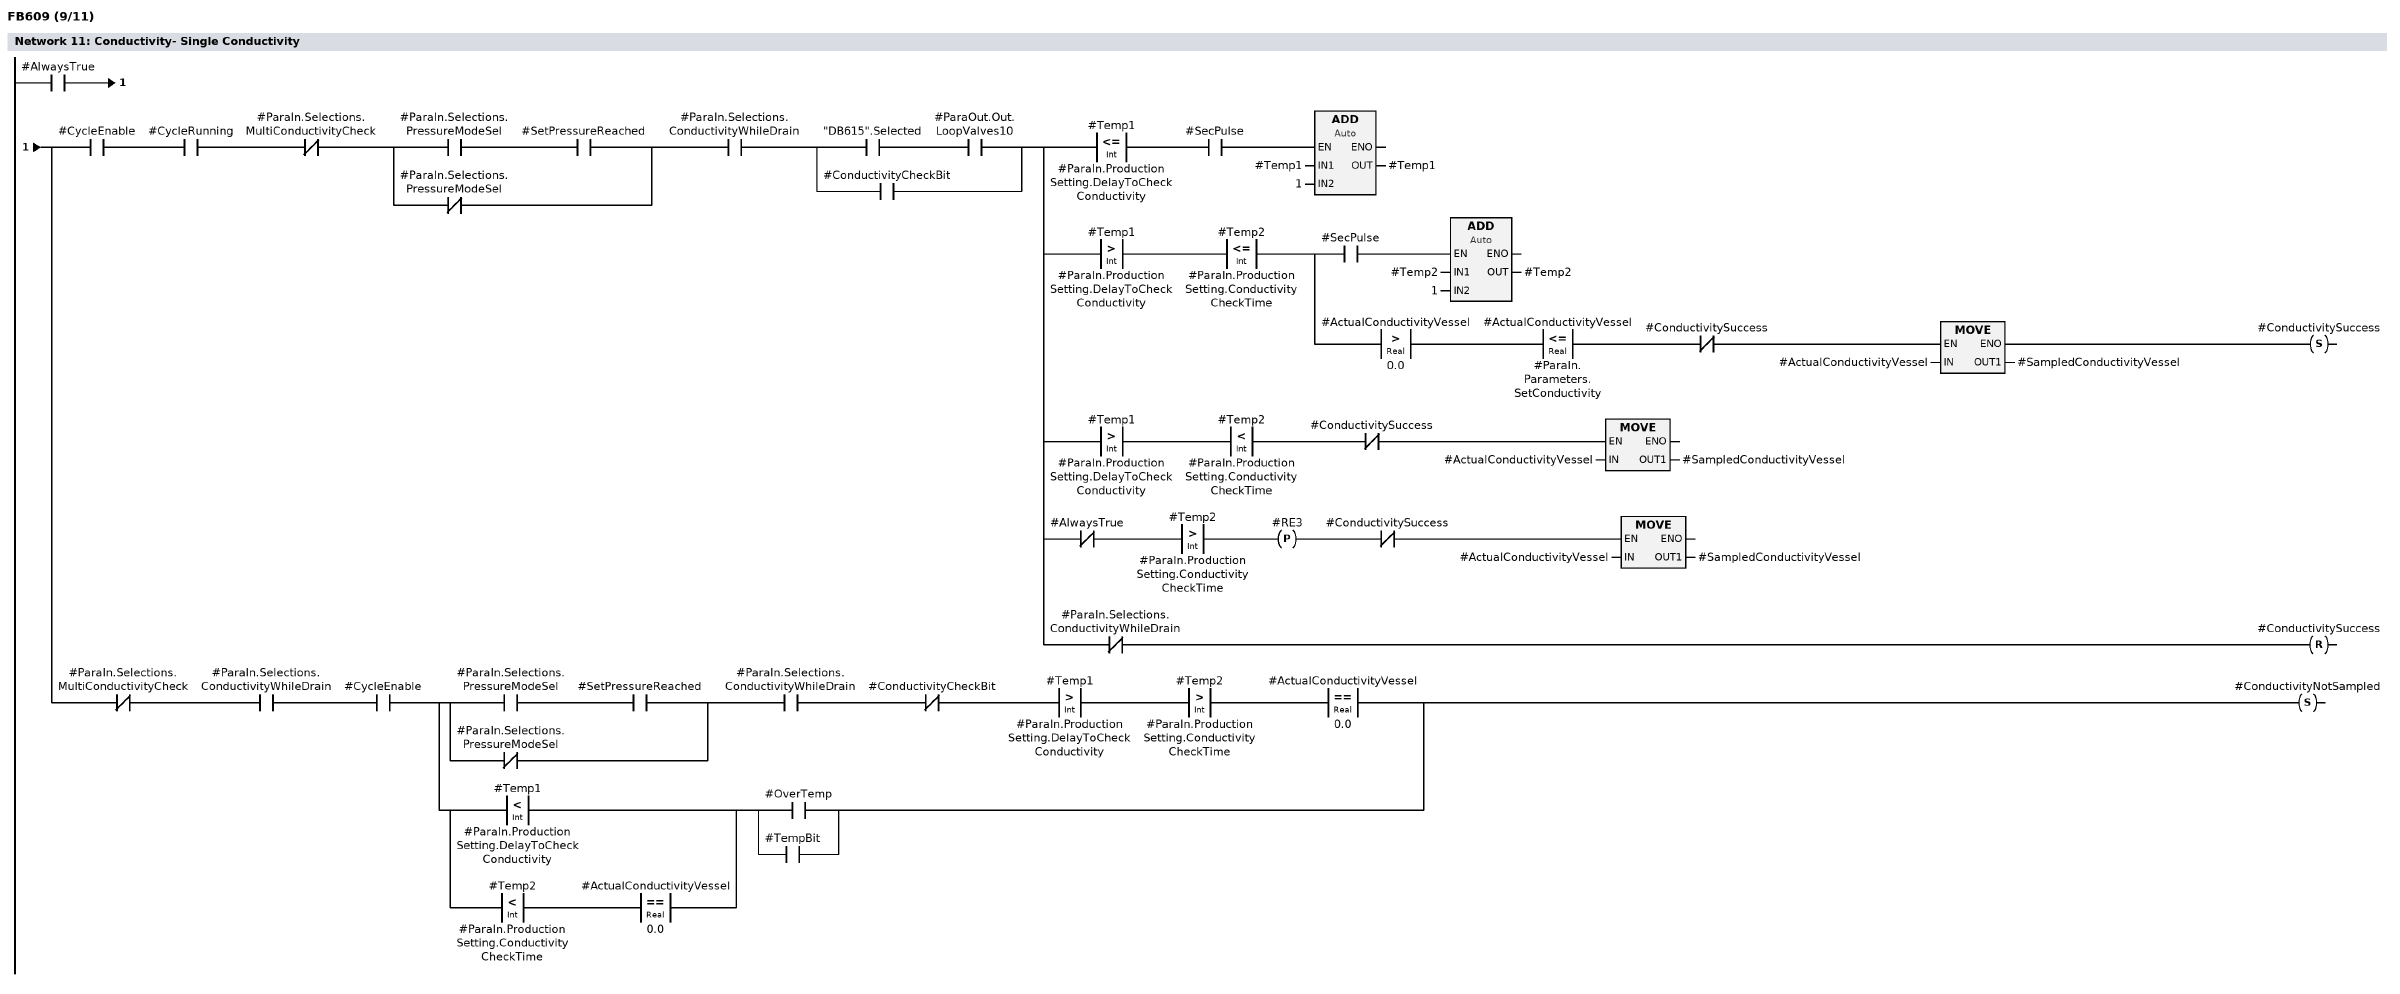
   RUNG wire#powerrail
      Contact( #AlwaysTrue )
      wire#w1
      Contact( #CycleEnable )
      Contact( #CycleRunning )
      I_Contact( #ParaIn.Selections.MultiConductivityCheck )
      wire#w2
      Contact( #ParaIn.Selections.PressureModeSel )
      Contact( #SetPressureReached )
      wire#w3
      Contact( #ParaIn.Selections.ConductivityWhileDrain )
      wire#w4
      Contact( "DB615".Selected )
      Contact( #ParaOut.Out.LoopValves10 )
      wire#w5
      { S7_Templates := "SrcType := Int" } LE_Contact(in1 := #Temp1, in2 := #ParaIn.ProductionSetting.DelayToCheckConductivity)
      Contact( #SecPulse )
      Add(in1 := #Temp1, in2 := 1, out => #Temp1)
   END_RUNG
   RUNG wire#w2
      I_Contact( #ParaIn.Selections.PressureModeSel )
   END_RUNG wire#w3
   RUNG wire#w4
      Contact( #ConductivityCheckBit )
   END_RUNG wire#w5
   RUNG wire#w5
      { S7_Templates := "SrcType := Int" } GT_Contact(in1 := #Temp1, in2 := #ParaIn.ProductionSetting.DelayToCheckConductivity)
      { S7_Templates := "SrcType := Int" } LE_Contact(in1 := #Temp2, in2 := #ParaIn.ProductionSetting.ConductivityCheckTime)
      wire#w6
      Contact( #SecPulse )
      Add(in1 := #Temp2, in2 := 1, out => #Temp2)
   END_RUNG
   RUNG wire#w6
      { S7_Templates := "SrcType := Real" } GT_Contact(in1 := #ActualConductivityVessel, in2 := 0.0)
      { S7_Templates := "SrcType := Real" } LE_Contact(in1 := #ActualConductivityVessel, in2 := #ParaIn.Parameters.SetConductivity)
      I_Contact( #ConductivitySuccess )
      Move(in := #ActualConductivityVessel, out1 => #SampledConductivityVessel)
      S_Coil( #ConductivitySuccess )
   END_RUNG
   RUNG wire#w5
      { S7_Templates := "SrcType := Int" } GT_Contact(in1 := #Temp1, in2 := #ParaIn.ProductionSetting.DelayToCheckConductivity)
      { S7_Templates := "SrcType := Int" } LT_Contact(in1 := #Temp2, in2 := #ParaIn.ProductionSetting.ConductivityCheckTime)
      I_Contact( #ConductivitySuccess )
      Move(in := #ActualConductivityVessel, out1 => #SampledConductivityVessel)
   END_RUNG
   RUNG wire#w5
      I_Contact( #AlwaysTrue )
      { S7_Templates := "SrcType := Int" } GT_Contact(in1 := #Temp2, in2 := #ParaIn.ProductionSetting.ConductivityCheckTime)
      P_Trig( #RE3 )
      I_Contact( #ConductivitySuccess )
      Move(in := #ActualConductivityVessel, out1 => #SampledConductivityVessel)
   END_RUNG
   RUNG wire#w5
      I_Contact( #ParaIn.Selections.ConductivityWhileDrain )
      R_Coil( #ConductivitySuccess )
   END_RUNG
   RUNG wire#w1
      I_Contact( #ParaIn.Selections.MultiConductivityCheck )
      Contact( #ParaIn.Selections.ConductivityWhileDrain )
      Contact( #CycleEnable )
      wire#w7
      Contact( #ParaIn.Selections.PressureModeSel )
      Contact( #SetPressureReached )
      wire#w8
      Contact( #ParaIn.Selections.ConductivityWhileDrain )
      I_Contact( #ConductivityCheckBit )
      { S7_Templates := "SrcType := Int" } GT_Contact(in1 := #Temp1, in2 := #ParaIn.ProductionSetting.DelayToCheckConductivity)
      { S7_Templates := "SrcType := Int" } GT_Contact(in1 := #Temp2, in2 := #ParaIn.ProductionSetting.ConductivityCheckTime)
      { S7_Templates := "SrcType := Real" } EQ_Contact(in1 := #ActualConductivityVessel, in2 := 0.0)
      wire#w9
      S_Coil( #ConductivityNotSampled )
   END_RUNG
   RUNG wire#w7
      I_Contact( #ParaIn.Selections.PressureModeSel )
   END_RUNG wire#w8
   RUNG wire#w7
      { S7_Templates := "SrcType := Int" } LT_Contact(in1 := #Temp1, in2 := #ParaIn.ProductionSetting.DelayToCheckConductivity)
      wire#w10
      Contact( #OverTemp )
   END_RUNG wire#w9
   RUNG wire#w7
      { S7_Templates := "SrcType := Int" } LT_Contact(in1 := #Temp2, in2 := #ParaIn.ProductionSetting.ConductivityCheckTime)
      { S7_Templates := "SrcType := Real" } EQ_Contact(in1 := #ActualConductivityVessel, in2 := 0.0)
   END_RUNG wire#w10
   RUNG wire#w10
      Contact( #TempBit )
   END_RUNG wire#w9
   // the same network as SCL:
   #_w1 := #AlwaysTrue AND #CycleEnable AND #CycleRunning AND NOT #ParaIn.Selections.MultiConductivityCheck AND ((#ParaIn.Selections.PressureModeSel AND #SetPressureReached) OR NOT #ParaIn.Selections.PressureModeSel) AND #ParaIn.Selections.ConductivityWhileDrain AND (("DB615".Selected AND #ParaOut.Out.LoopValves10) OR #ConductivityCheckBit);
   IF #_w1 AND (#Temp1 <= #ParaIn.ProductionSetting.DelayToCheckConductivity) AND #SecPulse THEN
       #Temp1 := #Temp1 + 1;
   END_IF;
   #_w2 := #_w1 AND (#Temp1 > #ParaIn.ProductionSetting.DelayToCheckConductivity) AND (#Temp2 <= #ParaIn.ProductionSetting.ConductivityCheckTime);
   IF #_w2 AND #SecPulse THEN #Temp2 := #Temp2 + 1; END_IF;
   IF #_w2 AND (#ActualConductivityVessel > 0.0) AND (#ActualConductivityVessel <= #ParaIn.Parameters.SetConductivity) AND NOT #ConductivitySuccess THEN
       #SampledConductivityVessel := #ActualConductivityVessel;
       #ConductivitySuccess := TRUE;
   END_IF;
   IF #_w1 AND (#Temp1 > #ParaIn.ProductionSetting.DelayToCheckConductivity) AND (#Temp2 < #ParaIn.ProductionSetting.ConductivityCheckTime) AND NOT #ConductivitySuccess THEN
       #SampledConductivityVessel := #ActualConductivityVessel;
   END_IF;
   #_w3 := #_w1 AND NOT #AlwaysTrue AND (#Temp2 > #ParaIn.ProductionSetting.ConductivityCheckTime);
   #_w4 := #_w3 AND NOT #RE3;   // rising edge
   #RE3 := #_w3;
   IF #_w4 AND NOT #ConductivitySuccess THEN #SampledConductivityVessel := #ActualConductivityVessel; END_IF;
   IF #_w1 AND NOT #ParaIn.Selections.ConductivityWhileDrain THEN #ConductivitySuccess := FALSE; END_IF;
   IF #AlwaysTrue AND NOT #ParaIn.Selections.MultiConductivityCheck AND #ParaIn.Selections.ConductivityWhileDrain AND #CycleEnable AND ((((#ParaIn.Selections.PressureModeSel AND #SetPressureReached) OR NOT #ParaIn.Selections.PressureModeSel) AND #ParaIn.Selections.ConductivityWhileDrain AND NOT #ConductivityCheckBit AND (#Temp1 > #ParaIn.ProductionSetting.DelayToCheckConductivity) AND (#Temp2 > #ParaIn.ProductionSetting.ConductivityCheckTime) AND (#ActualConductivityVessel = 0.0)) OR (((#Temp1 < #ParaIn.ProductionSetting.DelayToCheckConductivity) OR ((#Temp2 < #ParaIn.ProductionSetting.ConductivityCheckTime) AND (#ActualConductivityVessel = 0.0))) AND (#OverTemp OR #TempBit))) THEN
       #ConductivityNotSampled := TRUE;
   END_IF;
END_REGION

REGION Network 12: Conductivity- Multi Conductivity
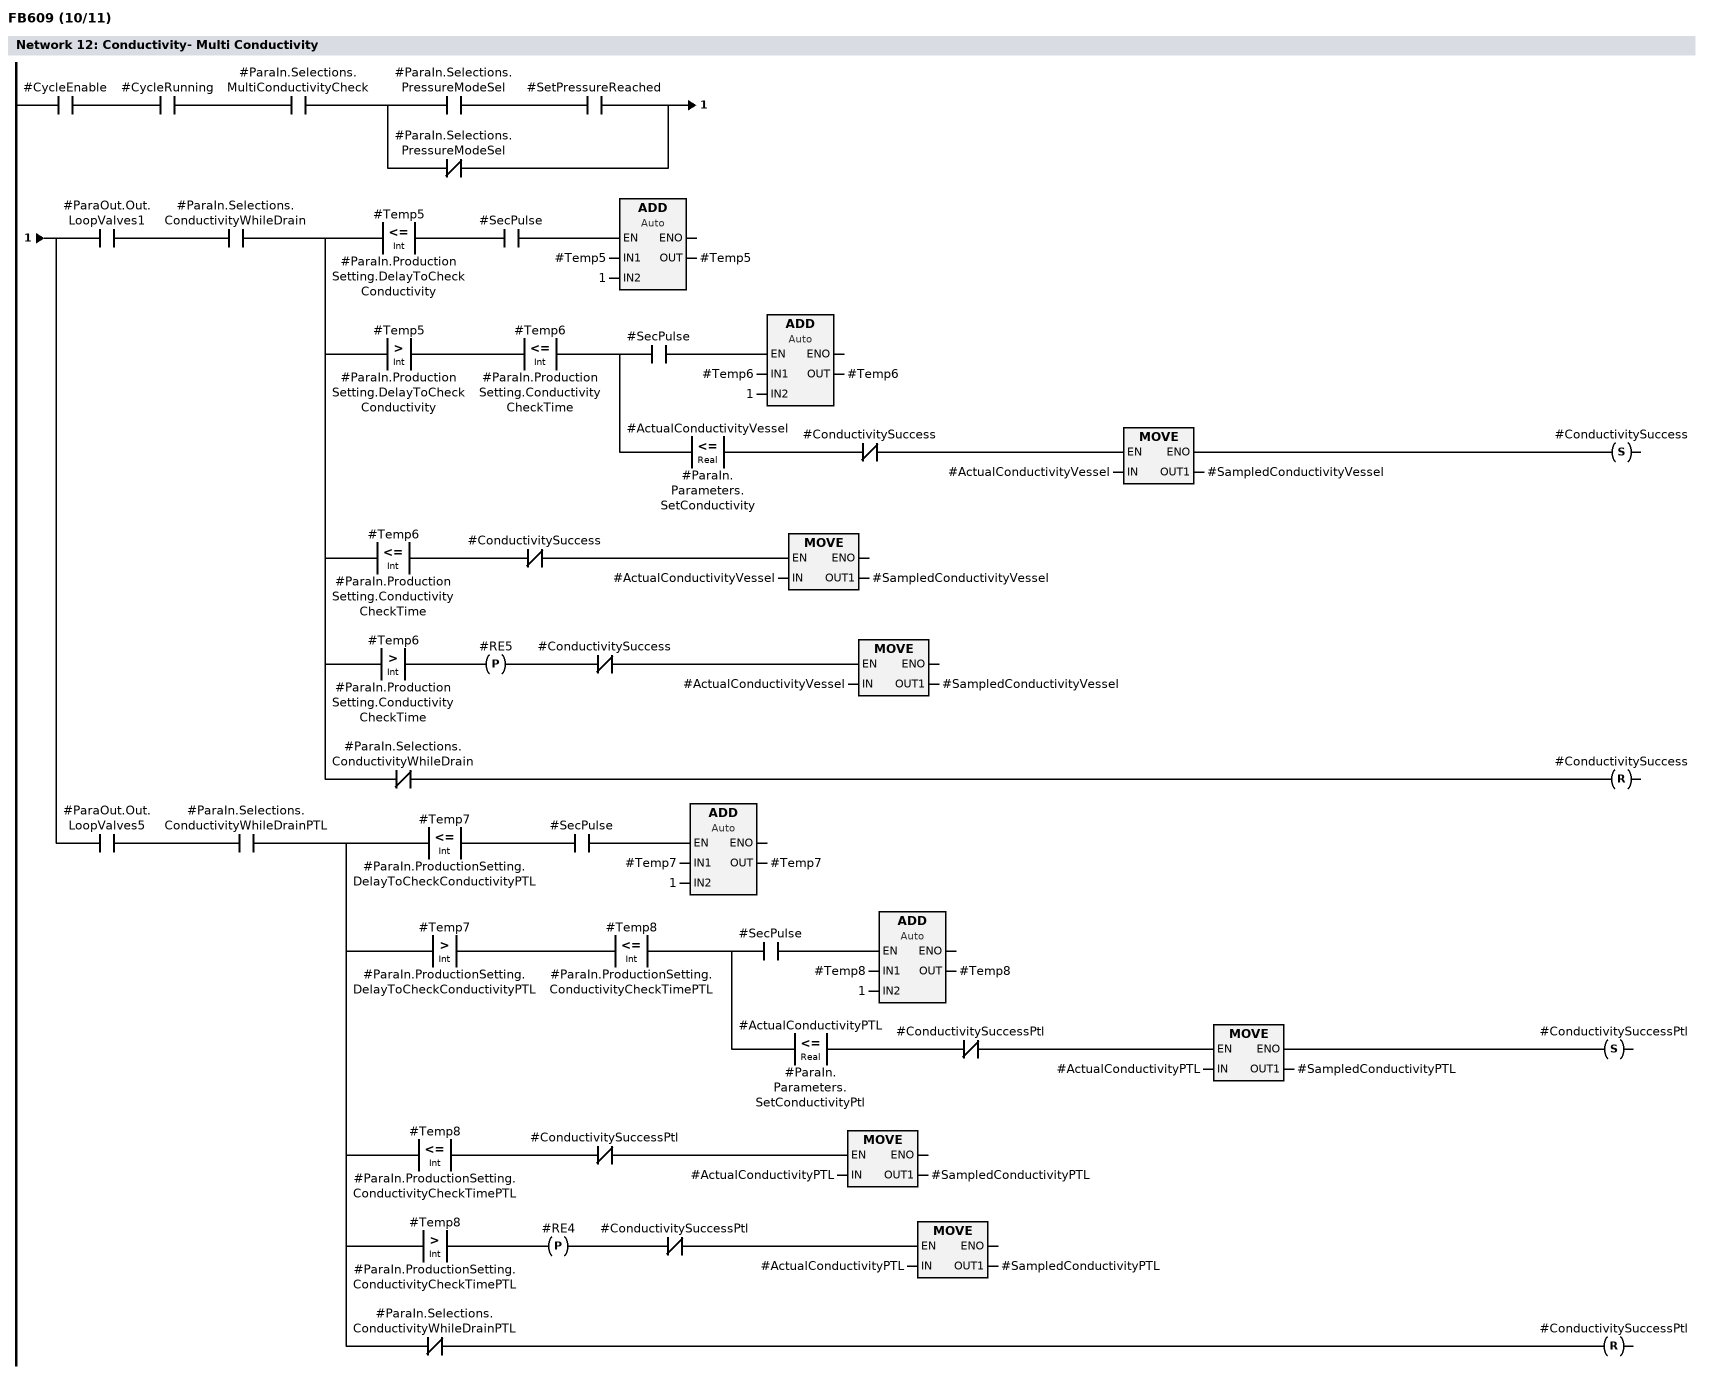
   RUNG wire#powerrail
      Contact( #CycleEnable )
      Contact( #CycleRunning )
      Contact( #ParaIn.Selections.MultiConductivityCheck )
      wire#w1
      Contact( #ParaIn.Selections.PressureModeSel )
      Contact( #SetPressureReached )
      wire#w2
      Contact( #ParaOut.Out.LoopValves1 )
      Contact( #ParaIn.Selections.ConductivityWhileDrain )
      wire#w3
      { S7_Templates := "SrcType := Int" } LE_Contact(in1 := #Temp5, in2 := #ParaIn.ProductionSetting.DelayToCheckConductivity)
      Contact( #SecPulse )
      Add(in1 := #Temp5, in2 := 1, out => #Temp5)
   END_RUNG
   RUNG wire#w1
      I_Contact( #ParaIn.Selections.PressureModeSel )
   END_RUNG wire#w2
   RUNG wire#w3
      { S7_Templates := "SrcType := Int" } GT_Contact(in1 := #Temp5, in2 := #ParaIn.ProductionSetting.DelayToCheckConductivity)
      { S7_Templates := "SrcType := Int" } LE_Contact(in1 := #Temp6, in2 := #ParaIn.ProductionSetting.ConductivityCheckTime)
      wire#w4
      Contact( #SecPulse )
      Add(in1 := #Temp6, in2 := 1, out => #Temp6)
   END_RUNG
   RUNG wire#w4
      { S7_Templates := "SrcType := Real" } LE_Contact(in1 := #ActualConductivityVessel, in2 := #ParaIn.Parameters.SetConductivity)
      I_Contact( #ConductivitySuccess )
      Move(in := #ActualConductivityVessel, out1 => #SampledConductivityVessel)
      S_Coil( #ConductivitySuccess )
   END_RUNG
   RUNG wire#w3
      { S7_Templates := "SrcType := Int" } LE_Contact(in1 := #Temp6, in2 := #ParaIn.ProductionSetting.ConductivityCheckTime)
      I_Contact( #ConductivitySuccess )
      Move(in := #ActualConductivityVessel, out1 => #SampledConductivityVessel)
   END_RUNG
   RUNG wire#w3
      { S7_Templates := "SrcType := Int" } GT_Contact(in1 := #Temp6, in2 := #ParaIn.ProductionSetting.ConductivityCheckTime)
      P_Trig( #RE5 )
      I_Contact( #ConductivitySuccess )
      Move(in := #ActualConductivityVessel, out1 => #SampledConductivityVessel)
   END_RUNG
   RUNG wire#w3
      I_Contact( #ParaIn.Selections.ConductivityWhileDrain )
      R_Coil( #ConductivitySuccess )
   END_RUNG
   RUNG wire#w2
      Contact( #ParaOut.Out.LoopValves5 )
      Contact( #ParaIn.Selections.ConductivityWhileDrainPTL )
      wire#w5
      { S7_Templates := "SrcType := Int" } LE_Contact(in1 := #Temp7, in2 := #ParaIn.ProductionSetting.DelayToCheckConductivityPTL)
      Contact( #SecPulse )
      Add(in1 := #Temp7, in2 := 1, out => #Temp7)
   END_RUNG
   RUNG wire#w5
      { S7_Templates := "SrcType := Int" } GT_Contact(in1 := #Temp7, in2 := #ParaIn.ProductionSetting.DelayToCheckConductivityPTL)
      { S7_Templates := "SrcType := Int" } LE_Contact(in1 := #Temp8, in2 := #ParaIn.ProductionSetting.ConductivityCheckTimePTL)
      wire#w6
      Contact( #SecPulse )
      Add(in1 := #Temp8, in2 := 1, out => #Temp8)
   END_RUNG
   RUNG wire#w6
      { S7_Templates := "SrcType := Real" } LE_Contact(in1 := #ActualConductivityPTL, in2 := #ParaIn.Parameters.SetConductivityPtl)
      I_Contact( #ConductivitySuccessPtl )
      Move(in := #ActualConductivityPTL, out1 => #SampledConductivityPTL)
      S_Coil( #ConductivitySuccessPtl )
   END_RUNG
   RUNG wire#w5
      { S7_Templates := "SrcType := Int" } LE_Contact(in1 := #Temp8, in2 := #ParaIn.ProductionSetting.ConductivityCheckTimePTL)
      I_Contact( #ConductivitySuccessPtl )
      Move(in := #ActualConductivityPTL, out1 => #SampledConductivityPTL)
   END_RUNG
   RUNG wire#w5
      { S7_Templates := "SrcType := Int" } GT_Contact(in1 := #Temp8, in2 := #ParaIn.ProductionSetting.ConductivityCheckTimePTL)
      P_Trig( #RE4 )
      I_Contact( #ConductivitySuccessPtl )
      Move(in := #ActualConductivityPTL, out1 => #SampledConductivityPTL)
   END_RUNG
   RUNG wire#w5
      I_Contact( #ParaIn.Selections.ConductivityWhileDrainPTL )
      R_Coil( #ConductivitySuccessPtl )
   END_RUNG
   // the same network as SCL:
   #_w1 := #CycleEnable AND #CycleRunning AND #ParaIn.Selections.MultiConductivityCheck AND ((#ParaIn.Selections.PressureModeSel AND #SetPressureReached) OR NOT #ParaIn.Selections.PressureModeSel);
   #_w2 := #_w1 AND #ParaOut.Out.LoopValves1 AND #ParaIn.Selections.ConductivityWhileDrain;
   IF #_w2 AND (#Temp5 <= #ParaIn.ProductionSetting.DelayToCheckConductivity) AND #SecPulse THEN
       #Temp5 := #Temp5 + 1;
   END_IF;
   #_w3 := #_w2 AND (#Temp5 > #ParaIn.ProductionSetting.DelayToCheckConductivity) AND (#Temp6 <= #ParaIn.ProductionSetting.ConductivityCheckTime);
   IF #_w3 AND #SecPulse THEN #Temp6 := #Temp6 + 1; END_IF;
   IF #_w3 AND (#ActualConductivityVessel <= #ParaIn.Parameters.SetConductivity) AND NOT #ConductivitySuccess THEN
       #SampledConductivityVessel := #ActualConductivityVessel;
       #ConductivitySuccess := TRUE;
   END_IF;
   IF #_w2 AND (#Temp6 <= #ParaIn.ProductionSetting.ConductivityCheckTime) AND NOT #ConductivitySuccess THEN
       #SampledConductivityVessel := #ActualConductivityVessel;
   END_IF;
   #_w4 := #_w2 AND (#Temp6 > #ParaIn.ProductionSetting.ConductivityCheckTime);
   #_w5 := #_w4 AND NOT #RE5;   // rising edge
   #RE5 := #_w4;
   IF #_w5 AND NOT #ConductivitySuccess THEN #SampledConductivityVessel := #ActualConductivityVessel; END_IF;
   IF #_w2 AND NOT #ParaIn.Selections.ConductivityWhileDrain THEN #ConductivitySuccess := FALSE; END_IF;
   #_w6 := #_w1 AND #ParaOut.Out.LoopValves5 AND #ParaIn.Selections.ConductivityWhileDrainPTL;
   IF #_w6 AND (#Temp7 <= #ParaIn.ProductionSetting.DelayToCheckConductivityPTL) AND #SecPulse THEN
       #Temp7 := #Temp7 + 1;
   END_IF;
   #_w7 := #_w6 AND (#Temp7 > #ParaIn.ProductionSetting.DelayToCheckConductivityPTL) AND (#Temp8 <= #ParaIn.ProductionSetting.ConductivityCheckTimePTL);
   IF #_w7 AND #SecPulse THEN #Temp8 := #Temp8 + 1; END_IF;
   IF #_w7 AND (#ActualConductivityPTL <= #ParaIn.Parameters.SetConductivityPtl) AND NOT #ConductivitySuccessPtl THEN
       #SampledConductivityPTL := #ActualConductivityPTL;
       #ConductivitySuccessPtl := TRUE;
   END_IF;
   IF #_w6 AND (#Temp8 <= #ParaIn.ProductionSetting.ConductivityCheckTimePTL) AND NOT #ConductivitySuccessPtl THEN
       #SampledConductivityPTL := #ActualConductivityPTL;
   END_IF;
   #_w8 := #_w6 AND (#Temp8 > #ParaIn.ProductionSetting.ConductivityCheckTimePTL);
   #_w9 := #_w8 AND NOT #RE4;   // rising edge
   #RE4 := #_w8;
   IF #_w9 AND NOT #ConductivitySuccessPtl THEN #SampledConductivityPTL := #ActualConductivityPTL; END_IF;
   IF #_w6 AND NOT #ParaIn.Selections.ConductivityWhileDrainPTL THEN
       #ConductivitySuccessPtl := FALSE;
   END_IF;
END_REGION

REGION Network 13: Reset Outputs
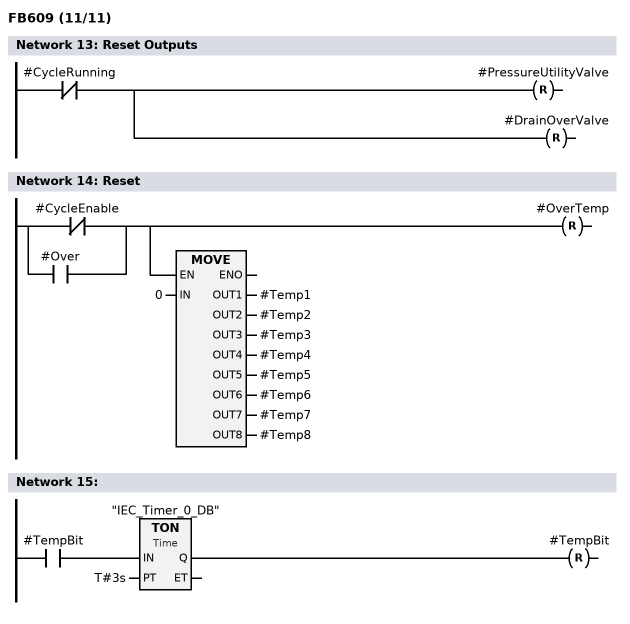
   RUNG wire#powerrail
      I_Contact( #CycleRunning )
      wire#w1
      R_Coil( #PressureUtilityValve )
   END_RUNG
   RUNG wire#w1
      R_Coil( #DrainOverValve )
   END_RUNG
   // the same network as SCL:
   IF NOT #CycleRunning THEN
       #PressureUtilityValve := FALSE;
       #DrainOverValve := FALSE;
   END_IF;
END_REGION

REGION Network 14: Reset
   RUNG wire#powerrail
      I_Contact( #CycleEnable )
      wire#w1
      R_Coil( #OverTemp )
   END_RUNG
   RUNG wire#powerrail
      Contact( #Over )
   END_RUNG wire#w1
   RUNG wire#w1
      Move(in := 0, out1 => #Temp1, out2 => #Temp2, out3 => #Temp3, out4 => #Temp4, out5 => #Temp5, out6 => #Temp6, out7 => #Temp7, out8 => #Temp8)
   END_RUNG
   // the same network as SCL:
   IF NOT #CycleEnable OR #Over THEN
       #OverTemp := FALSE;
       #Temp1 := 0;
       #Temp2 := 0;
       #Temp3 := 0;
       #Temp4 := 0;
       #Temp5 := 0;
       #Temp6 := 0;
       #Temp7 := 0;
       #Temp8 := 0;
   END_IF;
END_REGION

REGION Network 15
   RUNG wire#powerrail
      Contact( #TempBit )
      { S7_Templates := "time_type := Time" } "IEC_Timer_0_DB".TON(pt := T#3s, et =>)
      R_Coil( #TempBit )
   END_RUNG
   // the same network as SCL:
   "IEC_Timer_0_DB".TON(IN := #TempBit, PT := T#3s);
   IF "IEC_Timer_0_DB".Q THEN #TempBit := FALSE; END_IF;
END_REGION
END_FUNCTION_BLOCK

FUNCTION_BLOCK "FB610"   // FB610, LAD
TITLE = FB610
{ S7_Optimized_Access := 'FALSE' }
AUTHOR : PRECISE
FAMILY : PRECISE
// CIP SYSTEM DRAIN
// stored: AutoNumber false, SetENOAutomatically false
   VAR_INPUT
      CycleEnable : Bool;
      CycleRunning : Bool;
      SecPulse : Bool;
      AlwaysTrue : Bool;
      SetTime : Int := 30;
      Loops : Int;
      DelayBetweenLoops : Int := 3;
   END_VAR
   VAR_OUTPUT
      Started : Bool;
      ParaOut : "SystemDrainOutputs";
      TimePv : DInt;
      StepStatus : String[60];
   END_VAR
   VAR_IN_OUT
      Over : Bool;
      OverTemp : Bool;
      Popup : Bool;
      PopupAck : Bool;
      PopUpSel : Bool;
   END_VAR
   VAR
      RE1 : Bool;
      "Timer" { S7_SetPoint := 'True'} : "FB101";
   END_VAR
   VAR_TEMP   // added for the SCL form of the ladder/FBD networks
      _w1 : Bool;
      _w2 : Bool;
      _w3 : Bool;
   END_VAR
BEGIN

REGION Network 1: SystemDrainStarted
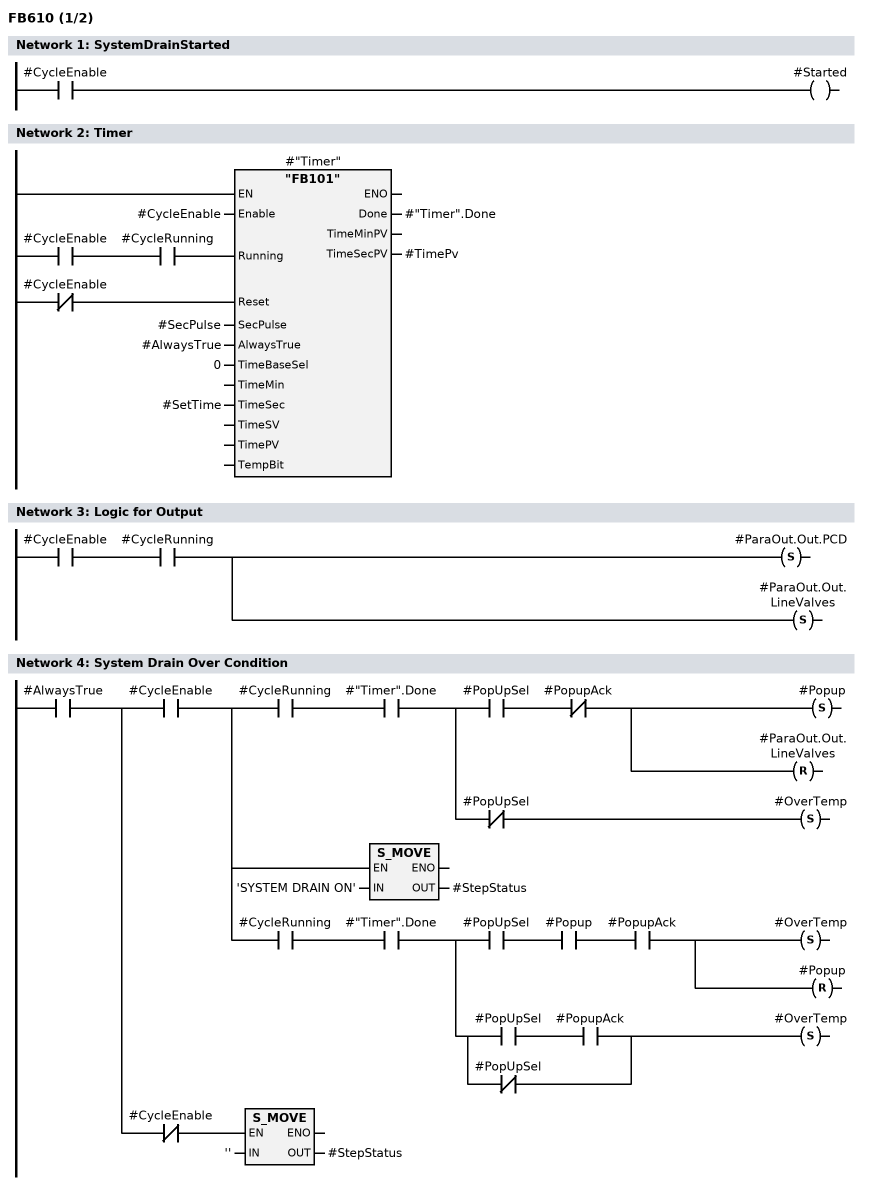
   RUNG wire#powerrail
      Contact( #CycleEnable )
      Coil( #Started )
   END_RUNG
   // the same network as SCL:
   #Started := #CycleEnable;
END_REGION

REGION Network 2: Timer
   RUNG wire#powerrail
      #"Timer"(Running := wire#w1, Reset := wire#w2, Enable := #CycleEnable, SecPulse := #SecPulse, AlwaysTrue := #AlwaysTrue, TimeBaseSel := 0, TimeMin :=, TimeSec := #SetTime, TimeSV :=, TimePV :=, TempBit :=, Done => #"Timer".Done, TimeMinPV =>, TimeSecPV => #TimePv)
   END_RUNG
   RUNG wire#powerrail
      Contact( #CycleEnable )
      Contact( #CycleRunning )
   END_RUNG wire#w1
   RUNG wire#powerrail
      I_Contact( #CycleEnable )
   END_RUNG wire#w2
   // the same network as SCL:
   #"Timer"(Enable := #CycleEnable,   // "FB101"
            Running := #CycleEnable AND #CycleRunning,
            Reset := NOT #CycleEnable,
            SecPulse := #SecPulse,
            AlwaysTrue := #AlwaysTrue,
            TimeBaseSel := 0,
            TimeSec := #SetTime,
            Done => #"Timer".Done,
            TimeSecPV => #TimePv);
END_REGION

REGION Network 3: Logic for Output
   RUNG wire#powerrail
      Contact( #CycleEnable )
      Contact( #CycleRunning )
      wire#w1
      S_Coil( #ParaOut.Out.PCD )
   END_RUNG
   RUNG wire#w1
      S_Coil( #ParaOut.Out.LineValves )
   END_RUNG
   // the same network as SCL:
   IF #CycleEnable AND #CycleRunning THEN
       #ParaOut.Out.PCD := TRUE;
       #ParaOut.Out.LineValves := TRUE;
   END_IF;
END_REGION

REGION Network 4: System Drain Over Condition
   RUNG wire#powerrail
      Contact( #AlwaysTrue )
      wire#w1
      Contact( #CycleEnable )
      wire#w2
      Contact( #CycleRunning )
      Contact( #"Timer".Done )
      wire#w3
      Contact( #PopUpSel )
      I_Contact( #PopupAck )
      wire#w4
      S_Coil( #Popup )
   END_RUNG
   RUNG wire#w4
      R_Coil( #ParaOut.Out.LineValves )
   END_RUNG
   RUNG wire#w3
      I_Contact( #PopUpSel )
      S_Coil( #OverTemp )
   END_RUNG
   RUNG wire#w2
      S_Move(in := 'SYSTEM DRAIN ON', out => #StepStatus)
   END_RUNG
   RUNG wire#w2
      Contact( #CycleRunning )
      Contact( #"Timer".Done )
      wire#w5
      Contact( #PopUpSel )
      Contact( #Popup )
      Contact( #PopupAck )
      wire#w6
      S_Coil( #OverTemp )
   END_RUNG
   RUNG wire#w6
      R_Coil( #Popup )
   END_RUNG
   RUNG wire#w5
      Contact( #PopUpSel )
      Contact( #PopupAck )
      wire#w7
      S_Coil( #OverTemp )
   END_RUNG
   RUNG wire#w5
      I_Contact( #PopUpSel )
   END_RUNG wire#w7
   RUNG wire#w1
      I_Contact( #CycleEnable )
      S_Move(in := '', out => #StepStatus)
   END_RUNG
   // the same network as SCL:
   #_w1 := #AlwaysTrue AND #CycleEnable;
   #_w2 := #_w1 AND #CycleRunning AND #"Timer".Done;
   IF #_w2 AND #PopUpSel AND NOT #PopupAck THEN
       #Popup := TRUE;
       #ParaOut.Out.LineValves := FALSE;
   END_IF;
   IF #_w2 AND NOT #PopUpSel THEN #OverTemp := TRUE; END_IF;
   IF #_w1 THEN #StepStatus := 'SYSTEM DRAIN ON'; END_IF;
   #_w3 := #_w1 AND #CycleRunning AND #"Timer".Done;
   IF #_w3 AND #PopUpSel AND #Popup AND #PopupAck THEN
       #OverTemp := TRUE;
       #Popup := FALSE;
   END_IF;
   IF #_w3 AND ((#PopUpSel AND #PopupAck) OR NOT #PopUpSel) THEN #OverTemp := TRUE; END_IF;
   IF #AlwaysTrue AND NOT #CycleEnable THEN #StepStatus := ''; END_IF;
END_REGION

REGION Network 5: System Drain Over
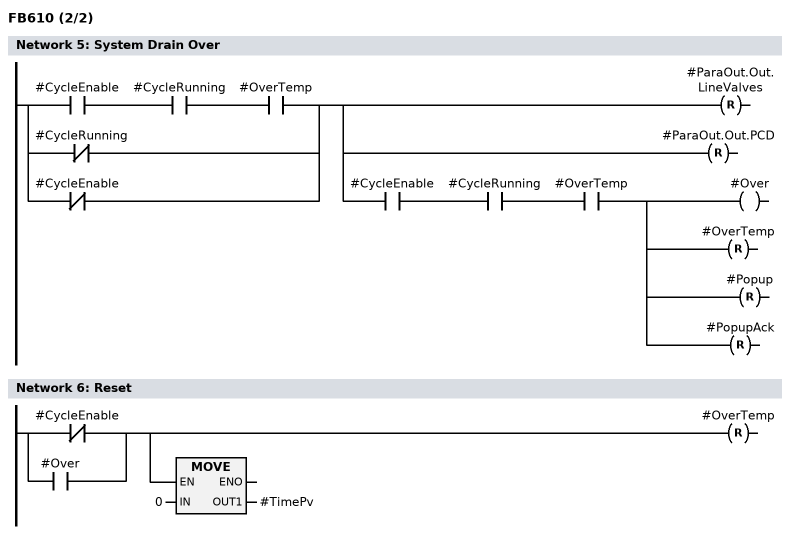
   RUNG wire#powerrail
      Contact( #CycleEnable )
      Contact( #CycleRunning )
      Contact( #OverTemp )
      wire#w1
      R_Coil( #ParaOut.Out.LineValves )
   END_RUNG
   RUNG wire#powerrail
      I_Contact( #CycleRunning )
   END_RUNG wire#w1
   RUNG wire#powerrail
      I_Contact( #CycleEnable )
   END_RUNG wire#w1
   RUNG wire#w1
      R_Coil( #ParaOut.Out.PCD )
   END_RUNG
   RUNG wire#w1
      Contact( #CycleEnable )
      Contact( #CycleRunning )
      Contact( #OverTemp )
      wire#w2
      Coil( #Over )
   END_RUNG
   RUNG wire#w2
      R_Coil( #OverTemp )
   END_RUNG
   RUNG wire#w2
      R_Coil( #Popup )
   END_RUNG
   RUNG wire#w2
      R_Coil( #PopupAck )
   END_RUNG
   // the same network as SCL:
   #_w1 := (#CycleEnable AND #CycleRunning AND #OverTemp) OR NOT #CycleRunning OR NOT #CycleEnable;
   IF #_w1 THEN
       #ParaOut.Out.LineValves := FALSE;
       #ParaOut.Out.PCD := FALSE;
   END_IF;
   #Over := #_w1 AND #CycleEnable AND #CycleRunning AND #OverTemp;
   IF #Over THEN
       #OverTemp := FALSE;
       #Popup := FALSE;
       #PopupAck := FALSE;
   END_IF;
END_REGION

REGION Network 6: Reset
   RUNG wire#powerrail
      I_Contact( #CycleEnable )
      wire#w1
      R_Coil( #OverTemp )
   END_RUNG
   RUNG wire#powerrail
      Contact( #Over )
   END_RUNG wire#w1
   RUNG wire#w1
      { S7_GenerateENO := "TRUE" } Move(in := 0, out1 => #TimePv)
   END_RUNG
   // the same network as SCL:
   IF NOT #CycleEnable OR #Over THEN
       #OverTemp := FALSE;
       #TimePv := 0;
   END_IF;
END_REGION
END_FUNCTION_BLOCK

FUNCTION_BLOCK "FB611"   // FB611, LAD
TITLE = FB611
{ S7_Optimized_Access := 'FALSE' }
AUTHOR : PRECISE
FAMILY : PRECISE
// CIP AIR PURGING
// stored: AutoNumber false, SetENOAutomatically false
   VAR_INPUT
      CycleEnable : Bool;
      CycleRunning : Bool;
      SecPulse : Bool;
      AlwaysTrue : Bool;
      ActualTemperature : Real;
      ActualPressure : Real;
      ActualRepetition : Int;
      ParaIn : "AirPurgingInputs";
   END_VAR
   VAR_OUTPUT
      Started : Bool;
      UtilityValve : Bool;   // Air Utility
      VentValve : Bool;
      ParaOut : "AirPurgingOutputs";
      StepStatus : String[60];
      TempValve : Bool;
      TempValve_close : Bool;
   END_VAR
   VAR_IN_OUT
      Over : Bool;
      OverTemp : Bool;
      PressurePostiveTol : Real;
      PressureNegativeTol : Real;
      ControlStarted : Bool;
      TempPostiveTol : Real;
      TempNegativeTol : Real;
      HotAirValve : Bool;
      PopupSel : Bool;
      Popup : Bool;
      PopupAck : Bool;
      ControlStartedTemp : Bool;
      re_5 : Bool;
      TempReached : Bool;
      re_6 : Bool;
   END_VAR
   VAR
      ValveOnDelayPV : Int;
      ValveOffDelayPV : Int;
      RE1 : Bool;
      StepDelay { S7_SetPoint := 'True'} : "FB110";
      VentTimer { S7_SetPoint := 'True'} : "FB101";
   END_VAR
   VAR_TEMP   // added for the SCL form of the ladder/FBD networks
      _w1 : Bool;
      _w2 : Bool;
      _w3 : Bool;
      _w4 : Bool;
   END_VAR
BEGIN

REGION Network 1: Air Purging Started
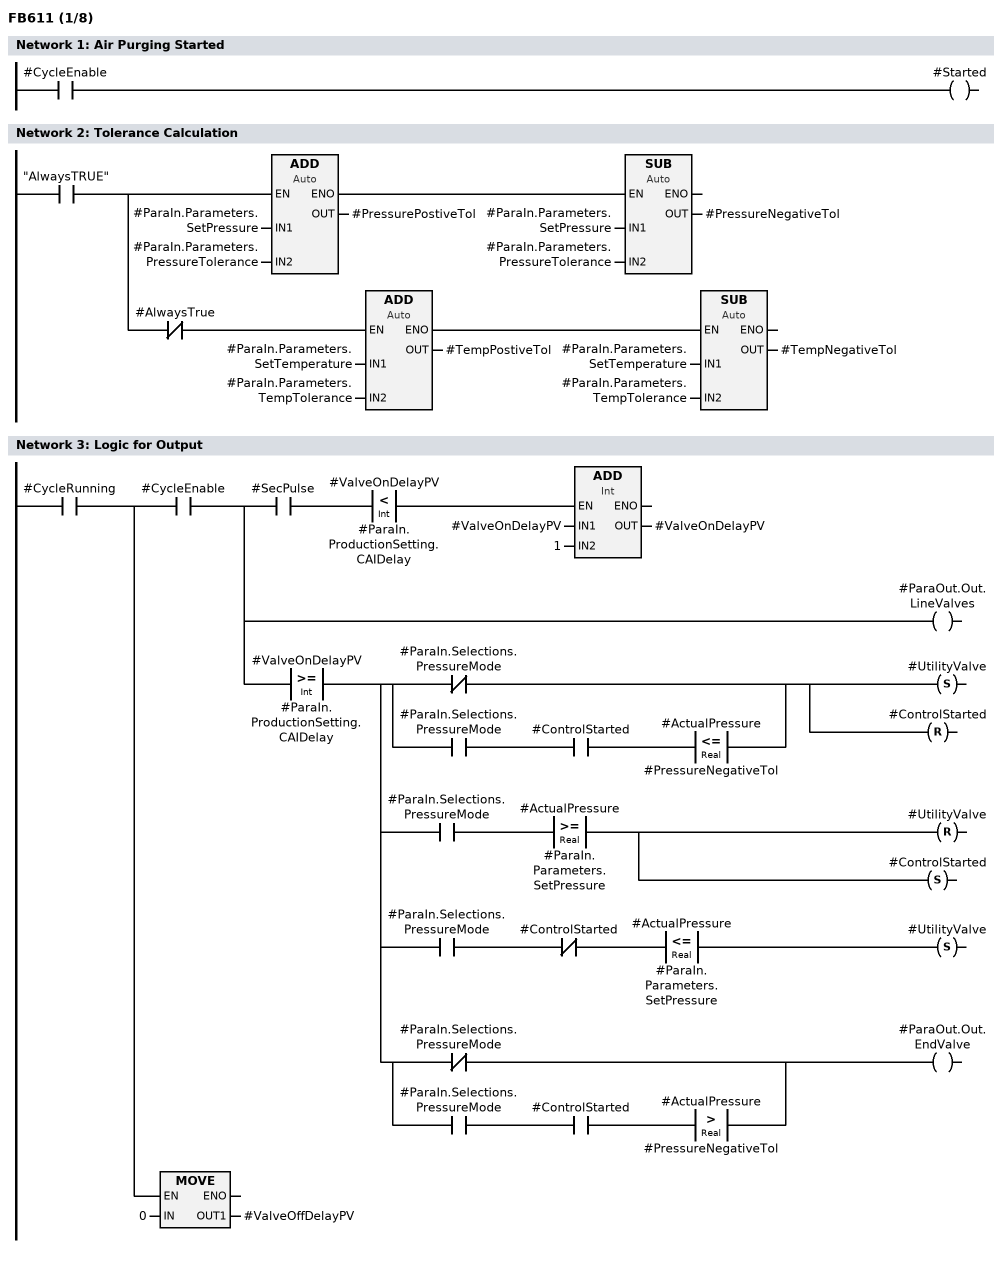
   RUNG wire#powerrail
      Contact( #CycleEnable )
      Coil( #Started )
   END_RUNG
   // the same network as SCL:
   #Started := #CycleEnable;
END_REGION

REGION Network 2: Tolerance Calculation
   RUNG wire#powerrail
      Contact( "AlwaysTRUE" )
      wire#w1
      Add(in1 := #ParaIn.Parameters.SetPressure, in2 := #ParaIn.Parameters.PressureTolerance, out => #PressurePostiveTol)
      Sub(in1 := #ParaIn.Parameters.SetPressure, in2 := #ParaIn.Parameters.PressureTolerance, out => #PressureNegativeTol)
   END_RUNG
   RUNG wire#w1
      I_Contact( #AlwaysTrue )
      Add(in1 := #ParaIn.Parameters.SetTemperature, in2 := #ParaIn.Parameters.TempTolerance, out => #TempPostiveTol)
      Sub(in1 := #ParaIn.Parameters.SetTemperature, in2 := #ParaIn.Parameters.TempTolerance, out => #TempNegativeTol)
   END_RUNG
   // the same network as SCL:
   IF "AlwaysTRUE" THEN
       #PressurePostiveTol := #ParaIn.Parameters.SetPressure + #ParaIn.Parameters.PressureTolerance;
       #PressureNegativeTol := #ParaIn.Parameters.SetPressure - #ParaIn.Parameters.PressureTolerance;
   END_IF;
   IF "AlwaysTRUE" AND NOT #AlwaysTrue THEN
       #TempPostiveTol := #ParaIn.Parameters.SetTemperature + #ParaIn.Parameters.TempTolerance;
       #TempNegativeTol := #ParaIn.Parameters.SetTemperature - #ParaIn.Parameters.TempTolerance;
   END_IF;
END_REGION

REGION Network 3: Logic for Output
   RUNG wire#powerrail
      Contact( #CycleRunning )
      wire#w1
      Contact( #CycleEnable )
      wire#w2
      Contact( #SecPulse )
      { S7_Templates := "SrcType := Int" } LT_Contact(in1 := #ValveOnDelayPV, in2 := #ParaIn.ProductionSetting.CAIDelay)
      { S7_Templates := "SrcType := Int"; S7_GenerateENO := "TRUE" } Add(in1 := #ValveOnDelayPV, in2 := 1, out => #ValveOnDelayPV)
   END_RUNG
   RUNG wire#w2
      Coil( #ParaOut.Out.LineValves )
   END_RUNG
   RUNG wire#w2
      { S7_Templates := "SrcType := Int" } GE_Contact(in1 := #ValveOnDelayPV, in2 := #ParaIn.ProductionSetting.CAIDelay)
      wire#w3
      I_Contact( #ParaIn.Selections.PressureMode )
      wire#w4
      S_Coil( #UtilityValve )
   END_RUNG
   RUNG wire#w3
      Contact( #ParaIn.Selections.PressureMode )
      Contact( #ControlStarted )
      { S7_Templates := "SrcType := Real" } LE_Contact(in1 := #ActualPressure, in2 := #PressureNegativeTol)
   END_RUNG wire#w4
   RUNG wire#w4
      R_Coil( #ControlStarted )
   END_RUNG
   RUNG wire#w3
      Contact( #ParaIn.Selections.PressureMode )
      { S7_Templates := "SrcType := Real" } GE_Contact(in1 := #ActualPressure, in2 := #ParaIn.Parameters.SetPressure)
      wire#w5
      R_Coil( #UtilityValve )
   END_RUNG
   RUNG wire#w5
      S_Coil( #ControlStarted )
   END_RUNG
   RUNG wire#w3
      Contact( #ParaIn.Selections.PressureMode )
      I_Contact( #ControlStarted )
      { S7_Templates := "SrcType := Real" } LE_Contact(in1 := #ActualPressure, in2 := #ParaIn.Parameters.SetPressure)
      S_Coil( #UtilityValve )
   END_RUNG
   RUNG wire#w3
      I_Contact( #ParaIn.Selections.PressureMode )
      wire#w6
      Coil( #ParaOut.Out.EndValve )
   END_RUNG
   RUNG wire#w3
      Contact( #ParaIn.Selections.PressureMode )
      Contact( #ControlStarted )
      { S7_Templates := "SrcType := Real" } GT_Contact(in1 := #ActualPressure, in2 := #PressureNegativeTol)
   END_RUNG wire#w6
   RUNG wire#w1
      { S7_GenerateENO := "TRUE" } Move(in := 0, out1 => #ValveOffDelayPV)
   END_RUNG
   // the same network as SCL:
   #_w1 := #CycleRunning AND #CycleEnable;
   IF #_w1 AND #SecPulse AND (#ValveOnDelayPV < #ParaIn.ProductionSetting.CAIDelay) THEN
       #ValveOnDelayPV := #ValveOnDelayPV + 1;
   END_IF;
   #ParaOut.Out.LineValves := #_w1;
   #_w2 := #_w1 AND (#ValveOnDelayPV >= #ParaIn.ProductionSetting.CAIDelay);
   IF #_w2 AND (NOT #ParaIn.Selections.PressureMode OR (#ParaIn.Selections.PressureMode AND #ControlStarted AND (#ActualPressure <= #PressureNegativeTol))) THEN
       #UtilityValve := TRUE;
       #ControlStarted := FALSE;
   END_IF;
   IF #_w2 AND #ParaIn.Selections.PressureMode AND (#ActualPressure >= #ParaIn.Parameters.SetPressure) THEN
       #UtilityValve := FALSE;
       #ControlStarted := TRUE;
   END_IF;
   IF #_w2 AND #ParaIn.Selections.PressureMode AND NOT #ControlStarted AND (#ActualPressure <= #ParaIn.Parameters.SetPressure) THEN
       #UtilityValve := TRUE;
   END_IF;
   #ParaOut.Out.EndValve := #_w2 AND (NOT #ParaIn.Selections.PressureMode OR (#ParaIn.Selections.PressureMode AND #ControlStarted AND (#ActualPressure > #PressureNegativeTol)));
   IF #CycleRunning THEN #ValveOffDelayPV := 0; END_IF;
END_REGION

REGION Network 4: Logic for Output Air Purging Sel
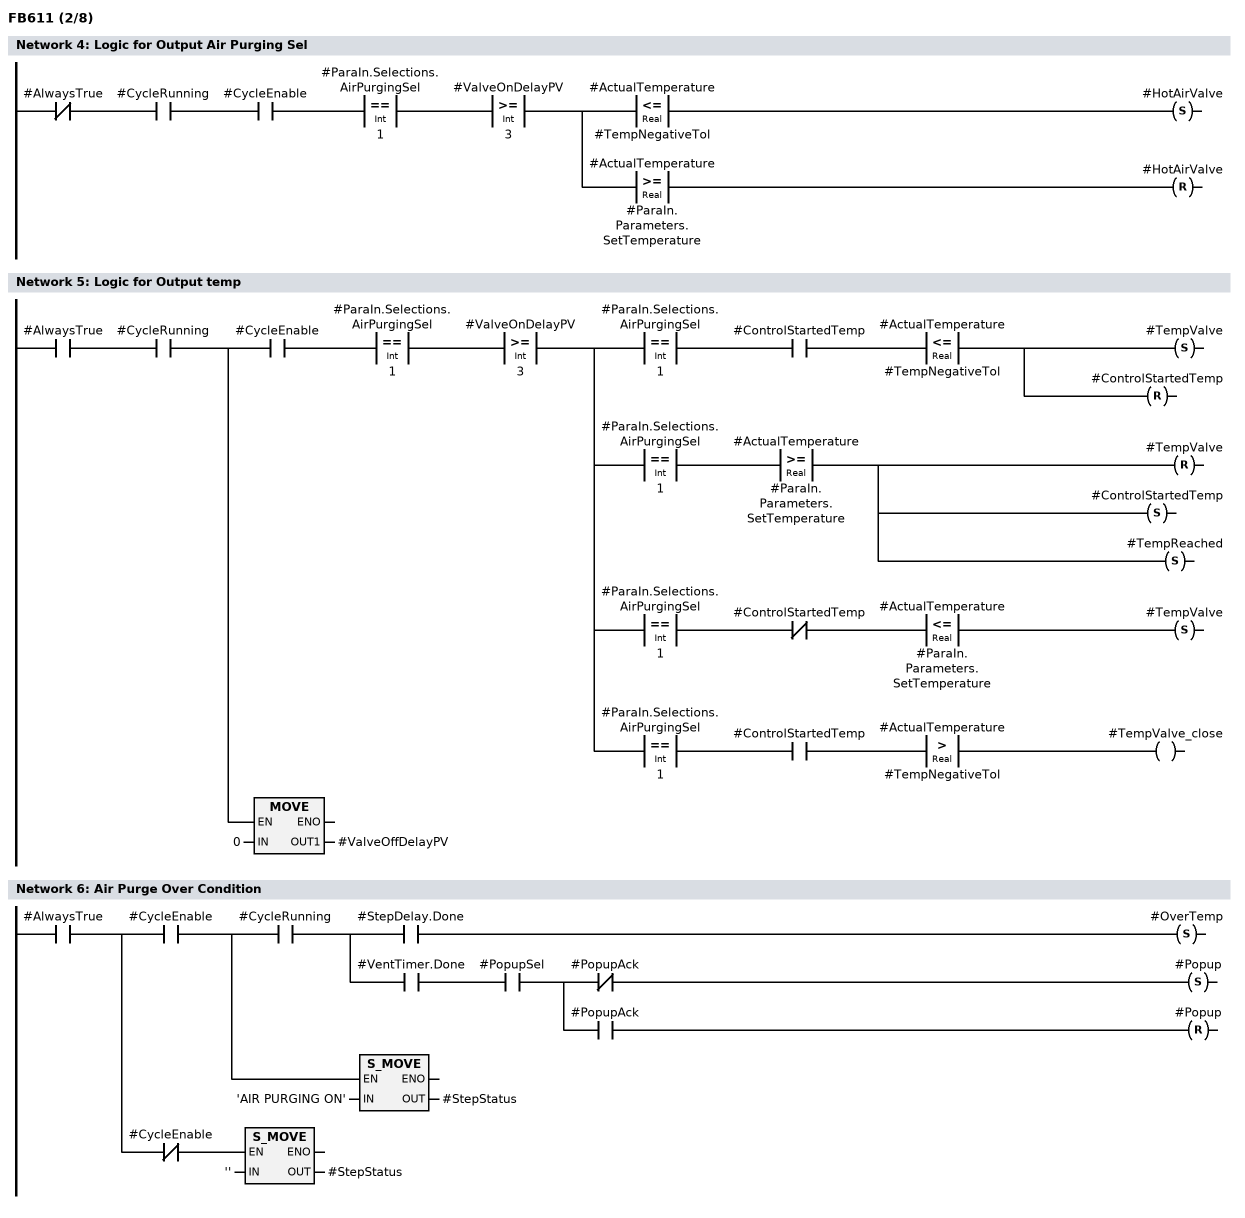
   RUNG wire#powerrail
      I_Contact( #AlwaysTrue )
      Contact( #CycleRunning )
      Contact( #CycleEnable )
      { S7_Templates := "SrcType := Int" } EQ_Contact(in1 := #ParaIn.Selections.AirPurgingSel, in2 := 1)
      { S7_Templates := "SrcType := Int" } GE_Contact(in1 := #ValveOnDelayPV, in2 := 3)
      wire#w1
      { S7_Templates := "SrcType := Real" } LE_Contact(in1 := #ActualTemperature, in2 := #TempNegativeTol)
      S_Coil( #HotAirValve )
   END_RUNG
   RUNG wire#w1
      { S7_Templates := "SrcType := Real" } GE_Contact(in1 := #ActualTemperature, in2 := #ParaIn.Parameters.SetTemperature)
      R_Coil( #HotAirValve )
   END_RUNG
   // the same network as SCL:
   #_w1 := NOT #AlwaysTrue AND #CycleRunning AND #CycleEnable AND (#ParaIn.Selections.AirPurgingSel = 1) AND (#ValveOnDelayPV >= 3);
   IF #_w1 AND (#ActualTemperature <= #TempNegativeTol) THEN #HotAirValve := TRUE; END_IF;
   IF #_w1 AND (#ActualTemperature >= #ParaIn.Parameters.SetTemperature) THEN #HotAirValve := FALSE; END_IF;
END_REGION

REGION Network 5: Logic for Output temp
   RUNG wire#powerrail
      Contact( #AlwaysTrue )
      Contact( #CycleRunning )
      wire#w1
      Contact( #CycleEnable )
      { S7_Templates := "SrcType := Int" } EQ_Contact(in1 := #ParaIn.Selections.AirPurgingSel, in2 := 1)
      { S7_Templates := "SrcType := Int" } GE_Contact(in1 := #ValveOnDelayPV, in2 := 3)
      wire#w2
      { S7_Templates := "SrcType := Int" } EQ_Contact(in1 := #ParaIn.Selections.AirPurgingSel, in2 := 1)
      Contact( #ControlStartedTemp )
      { S7_Templates := "SrcType := Real" } LE_Contact(in1 := #ActualTemperature, in2 := #TempNegativeTol)
      wire#w3
      S_Coil( #TempValve )
   END_RUNG
   RUNG wire#w3
      R_Coil( #ControlStartedTemp )
   END_RUNG
   RUNG wire#w2
      { S7_Templates := "SrcType := Int" } EQ_Contact(in1 := #ParaIn.Selections.AirPurgingSel, in2 := 1)
      { S7_Templates := "SrcType := Real" } GE_Contact(in1 := #ActualTemperature, in2 := #ParaIn.Parameters.SetTemperature)
      wire#w4
      R_Coil( #TempValve )
   END_RUNG
   RUNG wire#w4
      S_Coil( #ControlStartedTemp )
   END_RUNG
   RUNG wire#w4
      S_Coil( #TempReached )
   END_RUNG
   RUNG wire#w2
      { S7_Templates := "SrcType := Int" } EQ_Contact(in1 := #ParaIn.Selections.AirPurgingSel, in2 := 1)
      I_Contact( #ControlStartedTemp )
      { S7_Templates := "SrcType := Real" } LE_Contact(in1 := #ActualTemperature, in2 := #ParaIn.Parameters.SetTemperature)
      S_Coil( #TempValve )
   END_RUNG
   RUNG wire#w2
      { S7_Templates := "SrcType := Int" } EQ_Contact(in1 := #ParaIn.Selections.AirPurgingSel, in2 := 1)
      Contact( #ControlStartedTemp )
      { S7_Templates := "SrcType := Real" } GT_Contact(in1 := #ActualTemperature, in2 := #TempNegativeTol)
      Coil( #TempValve_close )
   END_RUNG
   RUNG wire#w1
      { S7_GenerateENO := "TRUE" } Move(in := 0, out1 => #ValveOffDelayPV)
   END_RUNG
   // the same network as SCL:
   #_w1 := #AlwaysTrue AND #CycleRunning;
   #_w2 := #_w1 AND #CycleEnable AND (#ParaIn.Selections.AirPurgingSel = 1) AND (#ValveOnDelayPV >= 3);
   IF #_w2 AND (#ParaIn.Selections.AirPurgingSel = 1) AND #ControlStartedTemp AND (#ActualTemperature <= #TempNegativeTol) THEN
       #TempValve := TRUE;
       #ControlStartedTemp := FALSE;
   END_IF;
   IF #_w2 AND (#ParaIn.Selections.AirPurgingSel = 1) AND (#ActualTemperature >= #ParaIn.Parameters.SetTemperature) THEN
       #TempValve := FALSE;
       #ControlStartedTemp := TRUE;
       #TempReached := TRUE;
   END_IF;
   IF #_w2 AND (#ParaIn.Selections.AirPurgingSel = 1) AND NOT #ControlStartedTemp AND (#ActualTemperature <= #ParaIn.Parameters.SetTemperature) THEN
       #TempValve := TRUE;
   END_IF;
   #TempValve_close := #_w2 AND (#ParaIn.Selections.AirPurgingSel = 1) AND #ControlStartedTemp AND (#ActualTemperature > #TempNegativeTol);
   IF #_w1 THEN #ValveOffDelayPV := 0; END_IF;
END_REGION

REGION Network 6: Air Purge Over Condition
   RUNG wire#powerrail
      Contact( #AlwaysTrue )
      wire#w1
      Contact( #CycleEnable )
      wire#w2
      Contact( #CycleRunning )
      wire#w3
      Contact( #StepDelay.Done )
      S_Coil( #OverTemp )
   END_RUNG
   RUNG wire#w3
      Contact( #VentTimer.Done )
      Contact( #PopupSel )
      wire#w4
      I_Contact( #PopupAck )
      S_Coil( #Popup )
   END_RUNG
   RUNG wire#w4
      Contact( #PopupAck )
      R_Coil( #Popup )
   END_RUNG
   RUNG wire#w2
      S_Move(in := 'AIR PURGING ON', out => #StepStatus)
   END_RUNG
   RUNG wire#w1
      I_Contact( #CycleEnable )
      S_Move(in := '', out => #StepStatus)
   END_RUNG
   // the same network as SCL:
   #_w1 := #AlwaysTrue AND #CycleEnable;
   #_w2 := #_w1 AND #CycleRunning;
   IF #_w2 AND #StepDelay.Done THEN #OverTemp := TRUE; END_IF;
   #_w3 := #_w2 AND #VentTimer.Done AND #PopupSel;
   IF #_w3 AND NOT #PopupAck THEN #Popup := TRUE; END_IF;
   IF #_w3 AND #PopupAck THEN #Popup := FALSE; END_IF;
   IF #_w1 THEN #StepStatus := 'AIR PURGING ON'; END_IF;
   IF #AlwaysTrue AND NOT #CycleEnable THEN #StepStatus := ''; END_IF;
END_REGION

REGION Network 7: Air Purge Over
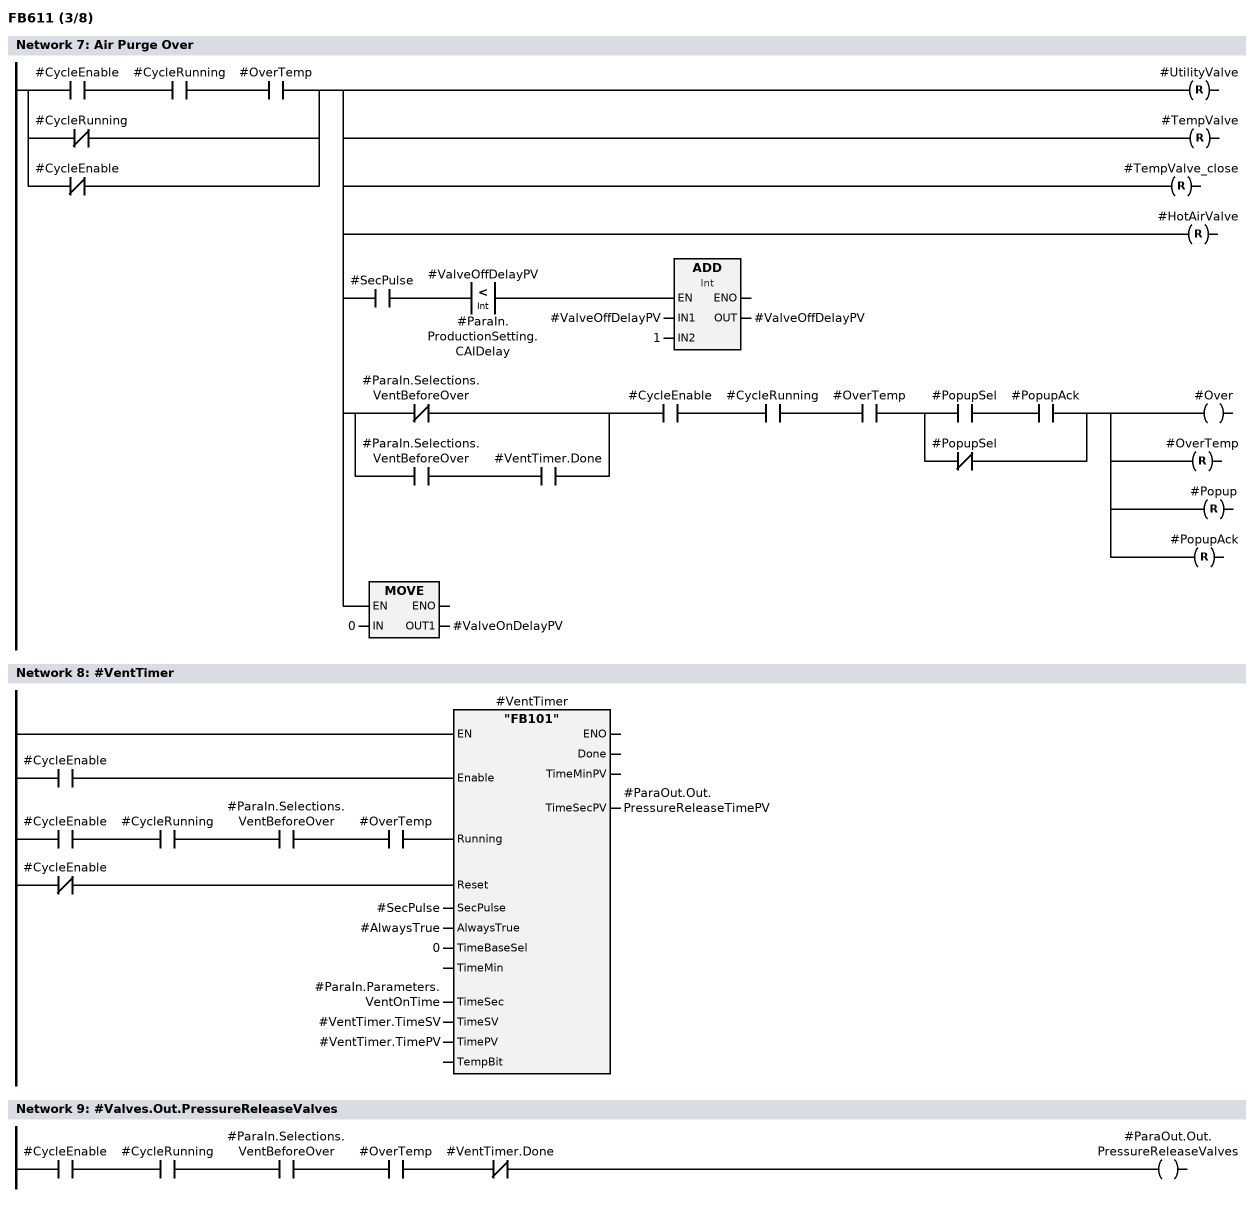
   RUNG wire#powerrail
      Contact( #CycleEnable )
      Contact( #CycleRunning )
      Contact( #OverTemp )
      wire#w1
      R_Coil( #UtilityValve )
   END_RUNG
   RUNG wire#powerrail
      I_Contact( #CycleRunning )
   END_RUNG wire#w1
   RUNG wire#powerrail
      I_Contact( #CycleEnable )
   END_RUNG wire#w1
   RUNG wire#w1
      R_Coil( #TempValve )
   END_RUNG
   RUNG wire#w1
      R_Coil( #TempValve_close )
   END_RUNG
   RUNG wire#w1
      R_Coil( #HotAirValve )
   END_RUNG
   RUNG wire#w1
      Contact( #SecPulse )
      { S7_Templates := "SrcType := Int" } LT_Contact(in1 := #ValveOffDelayPV, in2 := #ParaIn.ProductionSetting.CAIDelay)
      { S7_Templates := "SrcType := Int"; S7_GenerateENO := "TRUE" } Add(in1 := #ValveOffDelayPV, in2 := 1, out => #ValveOffDelayPV)
   END_RUNG
   RUNG wire#w1
      I_Contact( #ParaIn.Selections.VentBeforeOver )
      wire#w2
      Contact( #CycleEnable )
      Contact( #CycleRunning )
      Contact( #OverTemp )
      wire#w3
      Contact( #PopupSel )
      Contact( #PopupAck )
      wire#w4
      Coil( #Over )
   END_RUNG
   RUNG wire#w1
      Contact( #ParaIn.Selections.VentBeforeOver )
      Contact( #VentTimer.Done )
   END_RUNG wire#w2
   RUNG wire#w3
      I_Contact( #PopupSel )
   END_RUNG wire#w4
   RUNG wire#w4
      R_Coil( #OverTemp )
   END_RUNG
   RUNG wire#w4
      R_Coil( #Popup )
   END_RUNG
   RUNG wire#w4
      R_Coil( #PopupAck )
   END_RUNG
   RUNG wire#w1
      { S7_GenerateENO := "TRUE" } Move(in := 0, out1 => #ValveOnDelayPV)
   END_RUNG
   // the same network as SCL:
   #_w1 := (#CycleEnable AND #CycleRunning AND #OverTemp) OR NOT #CycleRunning OR NOT #CycleEnable;
   IF #_w1 THEN
       #UtilityValve := FALSE;
       #TempValve := FALSE;
       #TempValve_close := FALSE;
       #HotAirValve := FALSE;
   END_IF;
   IF #_w1 AND #SecPulse AND (#ValveOffDelayPV < #ParaIn.ProductionSetting.CAIDelay) THEN
       #ValveOffDelayPV := #ValveOffDelayPV + 1;
   END_IF;
   #Over := #_w1 AND (NOT #ParaIn.Selections.VentBeforeOver OR (#ParaIn.Selections.VentBeforeOver AND #VentTimer.Done)) AND #CycleEnable AND #CycleRunning AND #OverTemp AND ((#PopupSel AND #PopupAck) OR NOT #PopupSel);
   IF #Over THEN
       #OverTemp := FALSE;
       #Popup := FALSE;
       #PopupAck := FALSE;
   END_IF;
   IF #_w1 THEN #ValveOnDelayPV := 0; END_IF;
END_REGION

REGION Network 8: #VentTimer
   RUNG wire#powerrail
      #VentTimer(Enable := wire#w1, Running := wire#w2, Reset := wire#w3, SecPulse := #SecPulse, AlwaysTrue := #AlwaysTrue, TimeBaseSel := 0, TimeMin :=, TimeSec := #ParaIn.Parameters.VentOnTime, TimeSV := #VentTimer.TimeSV, TimePV := #VentTimer.TimePV, TempBit :=, Done =>, TimeMinPV =>, TimeSecPV => #ParaOut.Out.PressureReleaseTimePV)
   END_RUNG
   RUNG wire#powerrail
      Contact( #CycleEnable )
   END_RUNG wire#w1
   RUNG wire#powerrail
      Contact( #CycleEnable )
      Contact( #CycleRunning )
      Contact( #ParaIn.Selections.VentBeforeOver )
      Contact( #OverTemp )
   END_RUNG wire#w2
   RUNG wire#powerrail
      I_Contact( #CycleEnable )
   END_RUNG wire#w3
   // the same network as SCL:
   #VentTimer(Enable := #CycleEnable,   // "FB101"
              Running := #CycleEnable AND #CycleRunning AND #ParaIn.Selections.VentBeforeOver AND #OverTemp,
              Reset := NOT #CycleEnable,
              SecPulse := #SecPulse,
              AlwaysTrue := #AlwaysTrue,
              TimeBaseSel := 0,
              TimeSec := #ParaIn.Parameters.VentOnTime,
              TimeSV := #VentTimer.TimeSV,
              TimePV := #VentTimer.TimePV,
              TimeSecPV => #ParaOut.Out.PressureReleaseTimePV);
END_REGION

REGION Network 9: #Valves.Out.PressureReleaseValves
   RUNG wire#powerrail
      Contact( #CycleEnable )
      Contact( #CycleRunning )
      Contact( #ParaIn.Selections.VentBeforeOver )
      Contact( #OverTemp )
      I_Contact( #VentTimer.Done )
      Coil( #ParaOut.Out.PressureReleaseValves )
   END_RUNG
   // the same network as SCL:
   #ParaOut.Out.PressureReleaseValves := #CycleEnable AND #CycleRunning AND #ParaIn.Selections.VentBeforeOver AND #OverTemp AND NOT #VentTimer.Done;
END_REGION

REGION Network 10: StepDelay.StepTimeSV
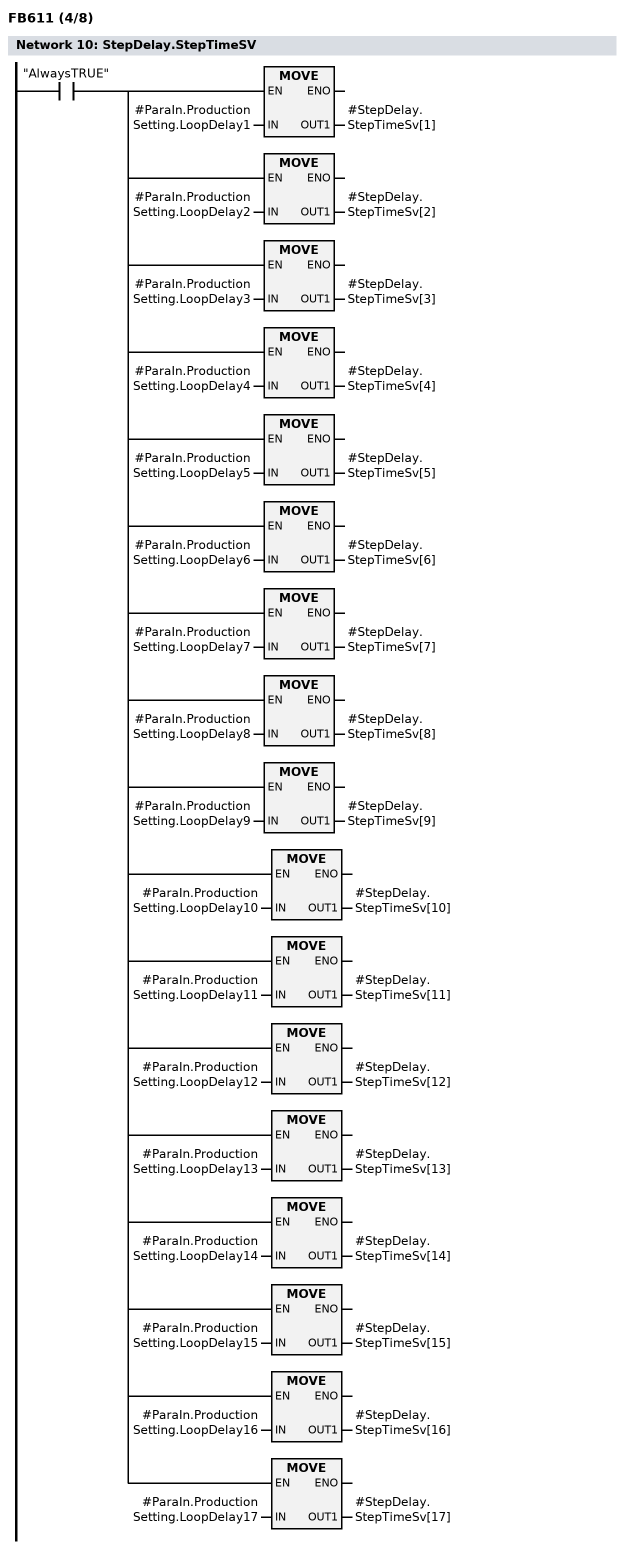
   RUNG wire#powerrail
      Contact( "AlwaysTRUE" )
      wire#w1
      Move(in := #ParaIn.ProductionSetting.LoopDelay1, out1 => #StepDelay.StepTimeSv[1])
   END_RUNG
   RUNG wire#w1
      Move(in := #ParaIn.ProductionSetting.LoopDelay2, out1 => #StepDelay.StepTimeSv[2])
   END_RUNG
   RUNG wire#w1
      Move(in := #ParaIn.ProductionSetting.LoopDelay3, out1 => #StepDelay.StepTimeSv[3])
   END_RUNG
   RUNG wire#w1
      Move(in := #ParaIn.ProductionSetting.LoopDelay4, out1 => #StepDelay.StepTimeSv[4])
   END_RUNG
   RUNG wire#w1
      Move(in := #ParaIn.ProductionSetting.LoopDelay5, out1 => #StepDelay.StepTimeSv[5])
   END_RUNG
   RUNG wire#w1
      Move(in := #ParaIn.ProductionSetting.LoopDelay6, out1 => #StepDelay.StepTimeSv[6])
   END_RUNG
   RUNG wire#w1
      Move(in := #ParaIn.ProductionSetting.LoopDelay7, out1 => #StepDelay.StepTimeSv[7])
   END_RUNG
   RUNG wire#w1
      Move(in := #ParaIn.ProductionSetting.LoopDelay8, out1 => #StepDelay.StepTimeSv[8])
   END_RUNG
   RUNG wire#w1
      Move(in := #ParaIn.ProductionSetting.LoopDelay9, out1 => #StepDelay.StepTimeSv[9])
   END_RUNG
   RUNG wire#w1
      Move(in := #ParaIn.ProductionSetting.LoopDelay10, out1 => #StepDelay.StepTimeSv[10])
   END_RUNG
   RUNG wire#w1
      Move(in := #ParaIn.ProductionSetting.LoopDelay11, out1 => #StepDelay.StepTimeSv[11])
   END_RUNG
   RUNG wire#w1
      Move(in := #ParaIn.ProductionSetting.LoopDelay12, out1 => #StepDelay.StepTimeSv[12])
   END_RUNG
   RUNG wire#w1
      Move(in := #ParaIn.ProductionSetting.LoopDelay13, out1 => #StepDelay.StepTimeSv[13])
   END_RUNG
   RUNG wire#w1
      Move(in := #ParaIn.ProductionSetting.LoopDelay14, out1 => #StepDelay.StepTimeSv[14])
   END_RUNG
   RUNG wire#w1
      Move(in := #ParaIn.ProductionSetting.LoopDelay15, out1 => #StepDelay.StepTimeSv[15])
   END_RUNG
   RUNG wire#w1
      Move(in := #ParaIn.ProductionSetting.LoopDelay16, out1 => #StepDelay.StepTimeSv[16])
   END_RUNG
   RUNG wire#w1
      Move(in := #ParaIn.ProductionSetting.LoopDelay17, out1 => #StepDelay.StepTimeSv[17])
   END_RUNG
   // the same network as SCL:
   IF "AlwaysTRUE" THEN
       #StepDelay.StepTimeSv[1] := #ParaIn.ProductionSetting.LoopDelay1;
       #StepDelay.StepTimeSv[2] := #ParaIn.ProductionSetting.LoopDelay2;
       #StepDelay.StepTimeSv[3] := #ParaIn.ProductionSetting.LoopDelay3;
       #StepDelay.StepTimeSv[4] := #ParaIn.ProductionSetting.LoopDelay4;
       #StepDelay.StepTimeSv[5] := #ParaIn.ProductionSetting.LoopDelay5;
       #StepDelay.StepTimeSv[6] := #ParaIn.ProductionSetting.LoopDelay6;
       #StepDelay.StepTimeSv[7] := #ParaIn.ProductionSetting.LoopDelay7;
       #StepDelay.StepTimeSv[8] := #ParaIn.ProductionSetting.LoopDelay8;
       #StepDelay.StepTimeSv[9] := #ParaIn.ProductionSetting.LoopDelay9;
       #StepDelay.StepTimeSv[10] := #ParaIn.ProductionSetting.LoopDelay10;
       #StepDelay.StepTimeSv[11] := #ParaIn.ProductionSetting.LoopDelay11;
       #StepDelay.StepTimeSv[12] := #ParaIn.ProductionSetting.LoopDelay12;
       #StepDelay.StepTimeSv[13] := #ParaIn.ProductionSetting.LoopDelay13;
       #StepDelay.StepTimeSv[14] := #ParaIn.ProductionSetting.LoopDelay14;
       #StepDelay.StepTimeSv[15] := #ParaIn.ProductionSetting.LoopDelay15;
       #StepDelay.StepTimeSv[16] := #ParaIn.ProductionSetting.LoopDelay16;
       #StepDelay.StepTimeSv[17] := #ParaIn.ProductionSetting.LoopDelay17;
   END_IF;
END_REGION

REGION Network 11: sv and pv for run screen
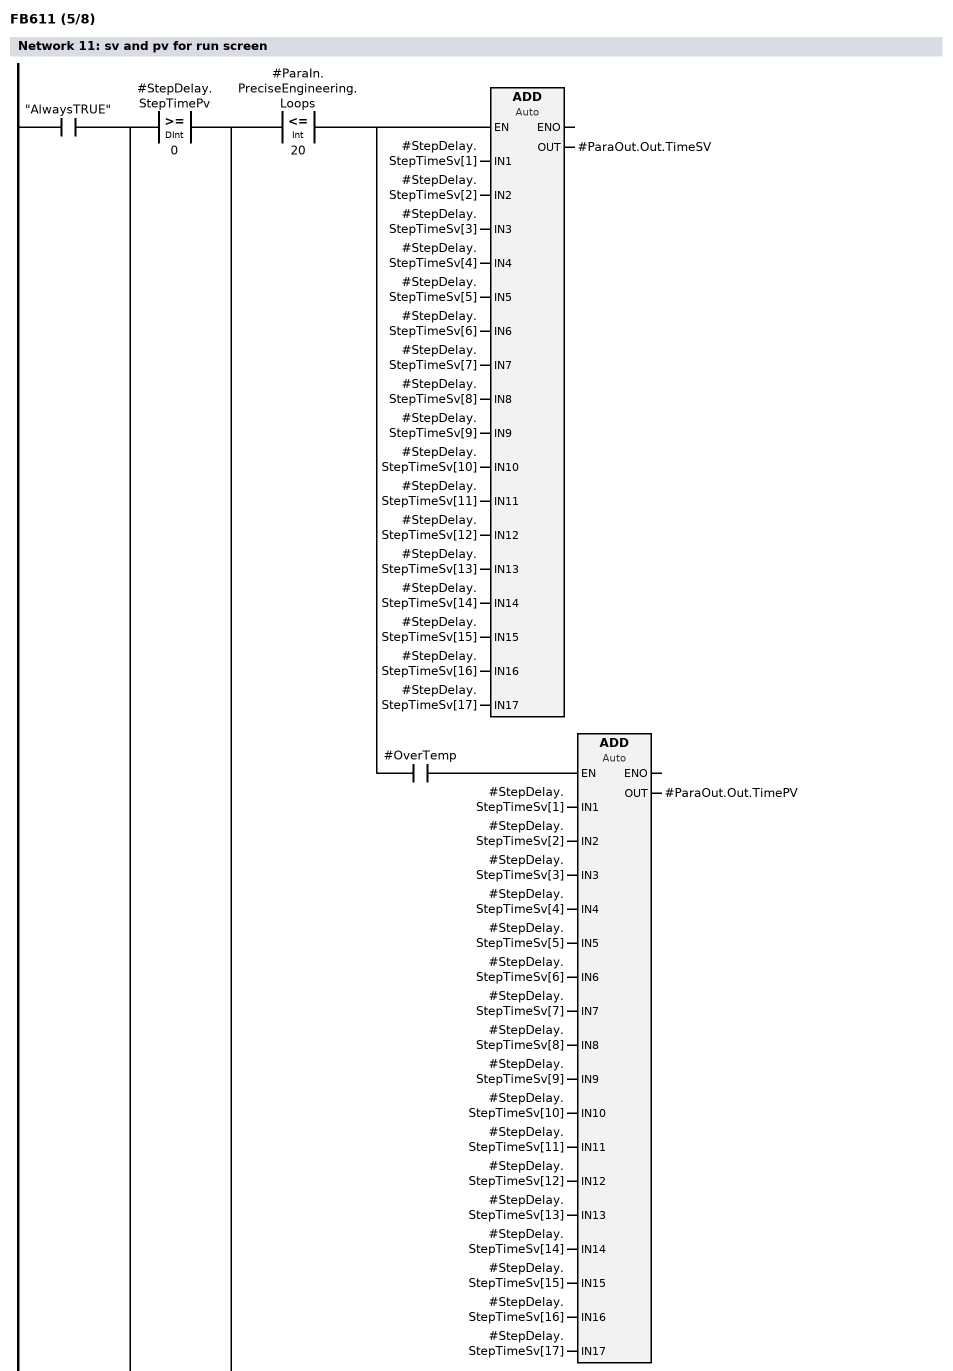
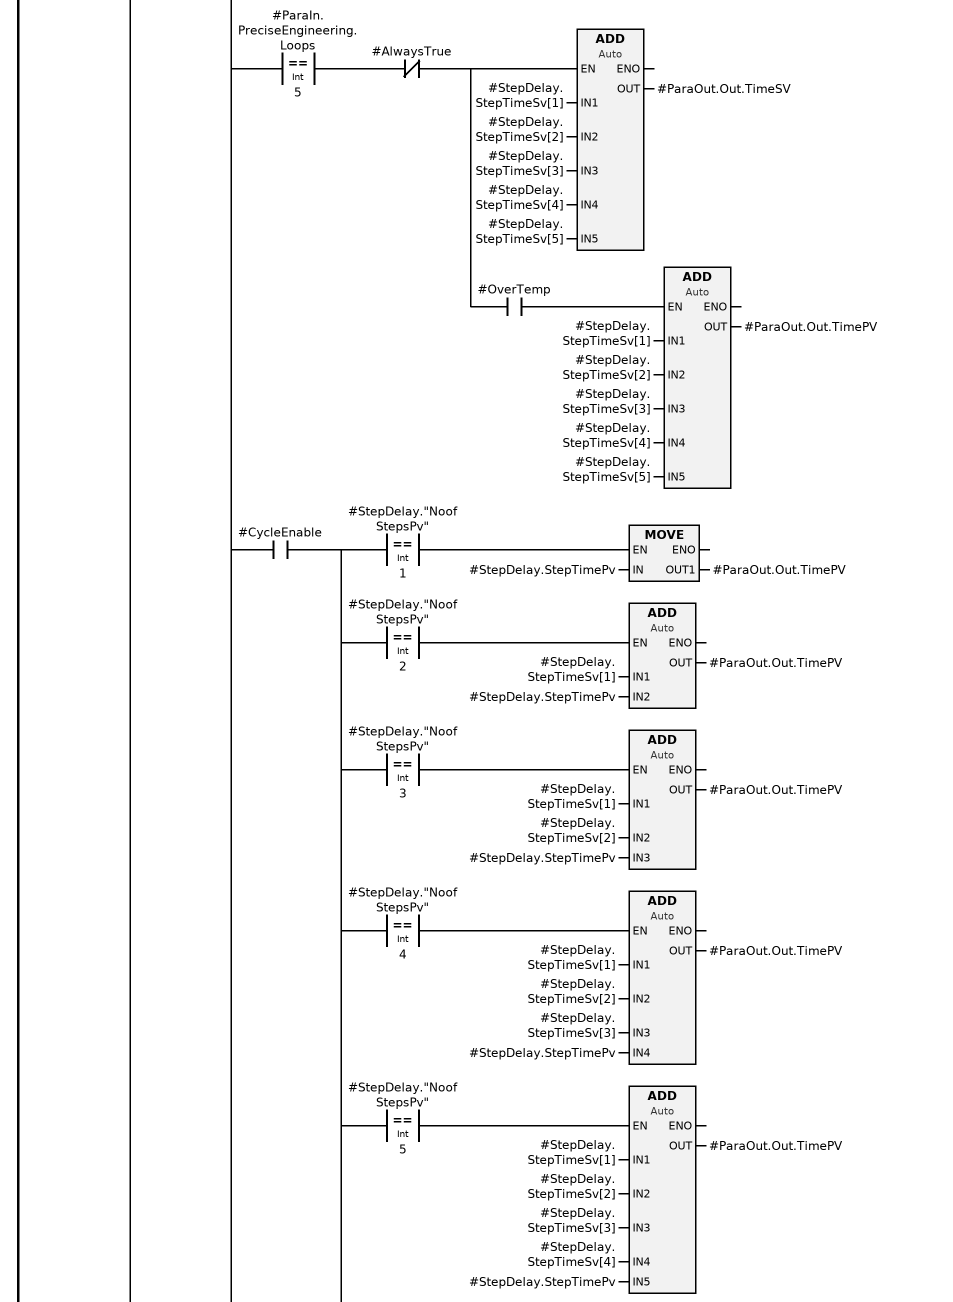
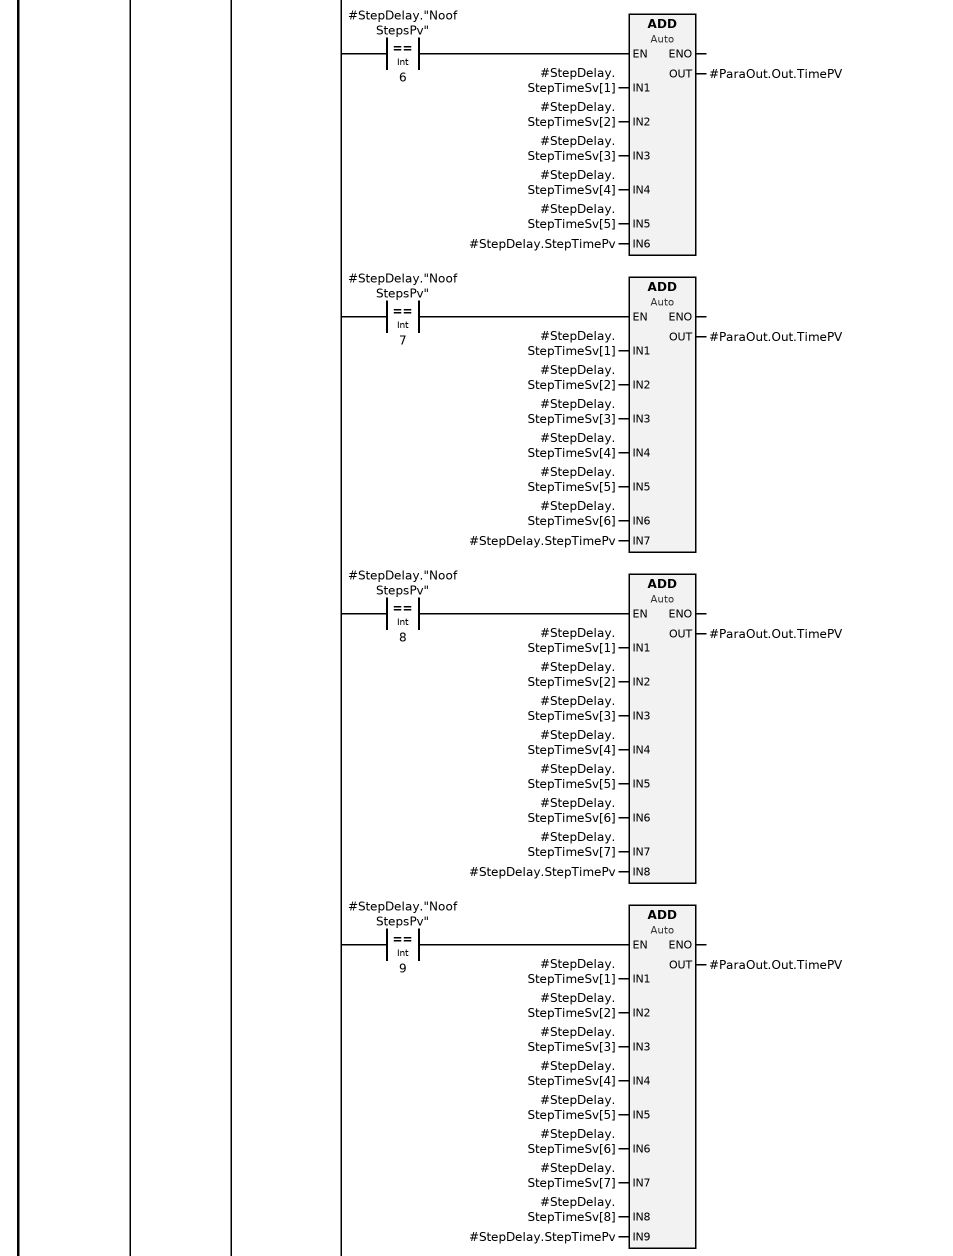
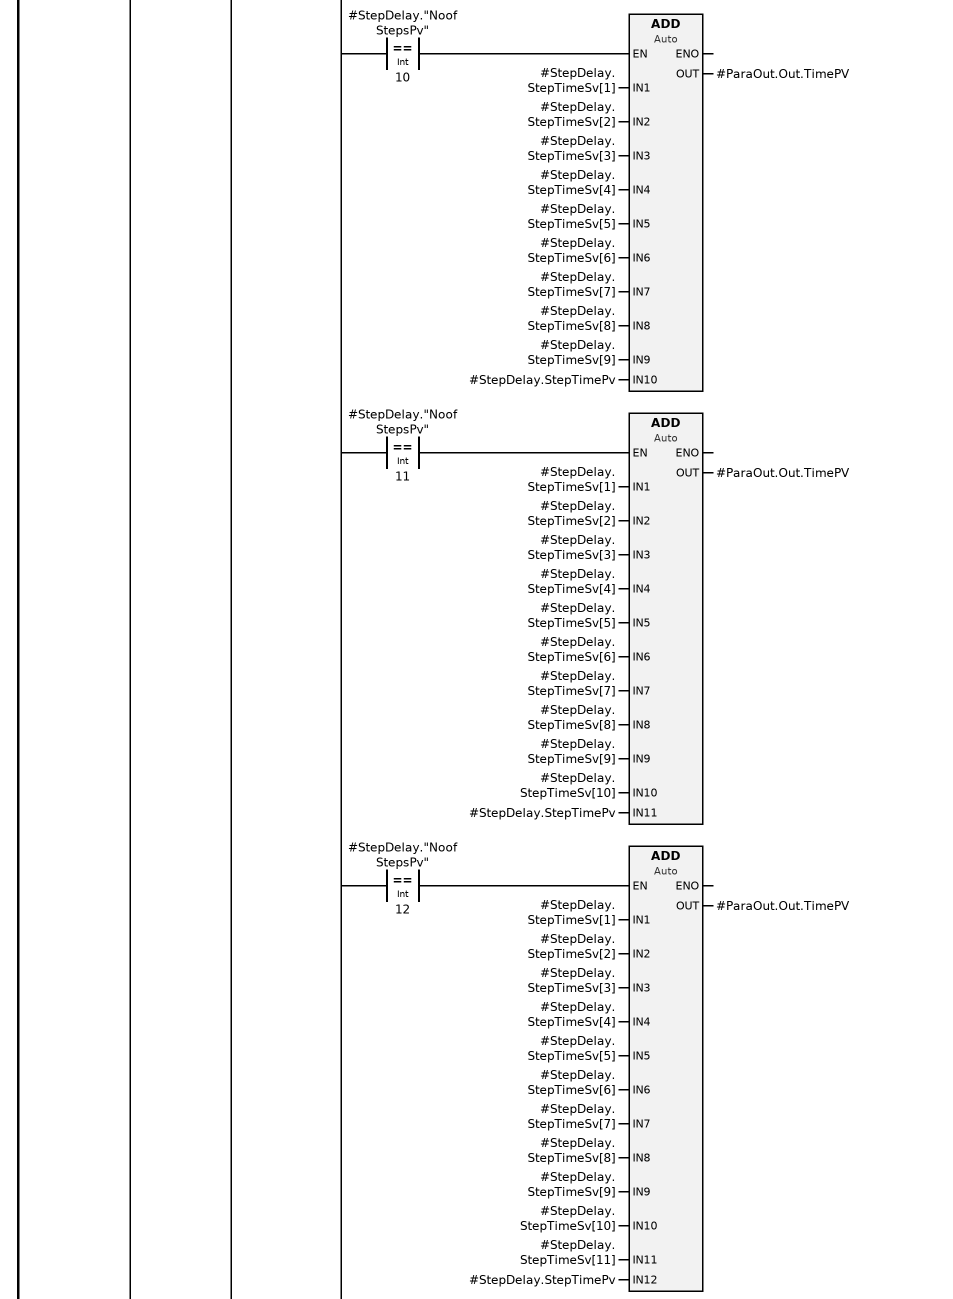
